TYPE "UDT_ConveyorInterface"
TITLE = UDT_ConveyorInterface
VERSION : 0.1
//User-defined structure of conveyor interface variables.
   STRUCT
      Displacement : Int;   // Displacement per PLC scan [cm] either from position (if available) or speed and time
      SpeedSetpoint : Int;   // Conveyor speed setpoint [mm/s]
      ActualSpeed : Int;   // Conveyors actual speed [mm/s]
      DeltaPosition : Int;   // Read from Conveyor Servo Position [mm] after 1 PLC cycle
      RunFwd { ExternalAccessible := 'False'; ExternalVisible := 'False'; ExternalWritable := 'False'} : Bool;   // Run forward request
      RunRvs { ExternalAccessible := 'False'; ExternalVisible := 'False'; ExternalWritable := 'False'} : Bool;   // Run reverse request
      InternalErrorEncoder { ExternalAccessible := 'False'; ExternalVisible := 'False'; ExternalWritable := 'False'} : Bool;   // Encoder has an error
      InternalErrorVFD { ExternalAccessible := 'False'; ExternalVisible := 'False'; ExternalWritable := 'False'} : Bool;   // VFD has an error
      InternalErrorTracking { ExternalAccessible := 'False'; ExternalVisible := 'False'; ExternalWritable := 'False'} : Bool;   // Tracking has an error
      InternalErrorPEC { ExternalAccessible := 'False'; ExternalVisible := 'False'; ExternalWritable := 'False'} : Bool;   // PEC has an error
      InternalWarningVFD { ExternalAccessible := 'False'; ExternalVisible := 'False'; ExternalWritable := 'False'} : Bool;   // VFD has a warning
      InternalWarningTracking { ExternalAccessible := 'False'; ExternalVisible := 'False'; ExternalWritable := 'False'} : Bool;   // Tracking has a warning
      InternalErrorReset { ExternalAccessible := 'False'; ExternalVisible := 'False'; ExternalWritable := 'False'} : Bool;   // Reset internal errors
      ConfigurationError { ExternalAccessible := 'False'; ExternalVisible := 'False'; ExternalWritable := 'False'} : Bool;   // Configuration error is active
      VFDRunning { ExternalAccessible := 'False'; ExternalVisible := 'False'; ExternalWritable := 'False'} : Bool;   // Motor is running
      VFDatSpeed { ExternalAccessible := 'False'; ExternalVisible := 'False'; ExternalWritable := 'False'} : Bool;   // Motor at speed setpoint
      Disconnected { ExternalAccessible := 'False'; ExternalVisible := 'False'; ExternalWritable := 'False'} : Bool;   // VFD disconnected
      ManualModeActive { ExternalAccessible := 'False'; ExternalVisible := 'False'; ExternalWritable := 'False'} : Bool;   // Covneyor is in manual mode
      ResetStatistics { ExternalAccessible := 'False'; ExternalVisible := 'False'; ExternalWritable := 'False'} : Bool;   // Reset statistics
      HardwareOk { ExternalAccessible := 'False'; ExternalVisible := 'False'; ExternalWritable := 'False'} : Bool;   // Hardware for the Equipment is available and healthy
   END_STRUCT;

END_TYPE

FUNCTION "FC_EquipmentReport" : Void
TITLE = FC_Equipment_Report
{ S7_Optimized_Access := 'TRUE' }
AUTHOR : MHSE
FAMILY : GeneralSystemFunctions
VERSION : 3.0
// ATTRIBUTES
// AUTO_NUMBER = True
// BLOCK_NUMBER = 16
// END_ATTRIBUTES
//Function to generate equipment report.
   VAR_INPUT
      iUDT_Status : "UDT_CommonStatus";   // Status structure
   END_VAR

   VAR_IN_OUT
      iqUDT_Control : "UDT_EquipmentControl";   // Equipment control
   END_VAR


BEGIN
	(*
	----------------------------------------------------------------------------------------

	Version history:
	Date        | Version   | Author        | Remark
	----------------------------------------------------------------------------------------
	24/05/2019  | 0.1       | F.Baten       | first release MHS TIA 15.1
	17/06/2019  | 0.3       | L.Klar        | Manual mode added to "UDT_EquipmentControl"
	17/07/2019  | 0.4       | A.Nowak       | Add all statuses and comments
	24/07/2019  | 2.0       | L.Klar        | 2.0 MHS library release TIA 15.1
	27/08/2019  | 2.1       | K.Pokorski    | Comments adjusted
	16/09/2019  | 2.2       | K.Pokorski    | Equipment error free condition added to "Restart required" status
	06/10/2019  | 2.3       | S. Deukar     | Updated accoring to new UDT equipment report
	12/11/2019  | 3.0       | P.Majka       | 3.0 MHS library release TIA 15.1
	05/02/2024  | 3.1       | L.Klar        | Auto On extention added
	13/03/2024  | 4.0       | S. Nieswiec   | Added to baseline
	*)

	REGION 1 - Equipment report update

	    // Extension of stopped equipment report with the stopped status
	    #iqUDT_Control.Report.Stopped := #iUDT_Status.Stopped
	    OR #iqUDT_Control.Report.Stopped;

	    // Extension of started equipment report with the started status
	    #iqUDT_Control.Report.Running := #iUDT_Status.Running
	    OR #iqUDT_Control.Report.Running;

	    // Extension of energy save equipment report with the energy save status
	    #iqUDT_Control.Report.EnergySave := #iUDT_Status.EnergySave
	    OR #iqUDT_Control.Report.EnergySave;

	    // Extension of warning equipment report with the warning status
	    #iqUDT_Control.Report.Warning := #iUDT_Status.Warning
	    OR #iqUDT_Control.Report.Warning;

	    // Extension of manual mode equipment report with the manual mode status
	    #iqUDT_Control.Report.Manual := #iUDT_Status.Manual
	    OR #iqUDT_Control.Report.Manual;

	    // Extension of error equipment report with the error status
	    #iqUDT_Control.Report.Error := #iUDT_Status.Error
	    OR #iqUDT_Control.Report.Error;

	    // Extension of safety stop equipment report with the safety stop status
	    #iqUDT_Control.Report.SafetyStop := #iUDT_Status.SafetyStop
	    OR #iqUDT_Control.Report.SafetyStop;

	    // Extension of Auto On equipment report with the Auto On status
	    #iqUDT_Control.Report.AutoON := #iUDT_Status.AutoON
	    OR #iqUDT_Control.Report.AutoON;

	    // Extension of restart required equipment report with the restart required and no equipment error statuses
	    #iqUDT_Control.Request.RestartRequired := #iUDT_Status.Stopped
	    AND NOT #iUDT_Status.Error
	    OR #iqUDT_Control.Request.RestartRequired;

	END_REGION
END_FUNCTION

TYPE "UDT_RIOStatistics"
TITLE = UDT_RIOStatistics
VERSION : 0.1
//User-defined structure of FB_RIO function block statistics.
   STRUCT
      PNSlaveNotOnline { S7_SetPoint := 'False'} : "UDT_EventStatistic";   // Statistics of  Profinet slave not online
      PNSlaveError { S7_SetPoint := 'False'} : "UDT_EventStatistic";   // Statistics of a Profinet slave error
   END_STRUCT;

END_TYPE

TYPE "UDT_FlowSplitterCommand"
TITLE = Flow Splitter Command
VERSION : 0.1
   STRUCT
      PercentageSplit : Int;   // Percentage value [%] that diverts are on.
      Mode : Int;   // 1- 100% transport; 2- 50% transport; 3- 100% divert; 4- % divert via HMI; 5- Semi automatic
      ManualMode { ExternalAccessible := 'False'; ExternalVisible := 'False'; ExternalWritable := 'False'} : Bool;   // Manual mode command from HMI
      ManualStartStop { ExternalAccessible := 'False'; ExternalVisible := 'False'; ExternalWritable := 'False'} : Bool;   // Start conveyor running when the bit is true, stop conveyor when the bit is false
      ManualFullSpeed { ExternalAccessible := 'False'; ExternalVisible := 'False'; ExternalWritable := 'False'} : Bool;   // Full speed conveyor in manual mode
      ManualJog { ExternalAccessible := 'False'; ExternalVisible := 'False'; ExternalWritable := 'False'} : Bool;   // Command to jog conveyor in slow speed from HMI
      Zone1DivertActivation { ExternalAccessible := 'False'; ExternalVisible := 'False'; ExternalWritable := 'False'} : Bool;   // Active diverts in zone 1
      Zone2DivertActivation { ExternalAccessible := 'False'; ExternalVisible := 'False'; ExternalWritable := 'False'} : Bool;   // Active diverts in zone 2
   END_STRUCT;

END_TYPE

TYPE "UDT_FlowSplitterStatus"
TITLE = Flow splitter status
VERSION : 0.1
   STRUCT
      Status : Int;   // Status number
      Specific : Struct
         Mode : Int;   // Mode: 1- 100% transport; 2- 50% transport; 3- 100% divert; 4- % divert via HMI; 5- Semi automatic
         Debris { ExternalAccessible := 'False'; ExternalVisible := 'False'; ExternalWritable := 'False'} : Bool;   // Debris detected under the belt
         PEC_EoSJam { ExternalAccessible := 'False'; ExternalVisible := 'False'; ExternalWritable := 'False'} : Bool;   // PEC Jam detected
         PEC_DivertChuteJam { ExternalAccessible := 'False'; ExternalVisible := 'False'; ExternalWritable := 'False'} : Bool;   // PEC divert chute jam detected
         DivertsActivationError { ExternalAccessible := 'False'; ExternalVisible := 'False'; ExternalWritable := 'False'} : Bool;   // Error when zone 1 is not active but zone 2 is active
         AirPressure { ExternalAccessible := 'False'; ExternalVisible := 'False'; ExternalWritable := 'False'} : Bool;   // Air pressure error
         EncoderError { ExternalAccessible := 'False'; ExternalVisible := 'False'; ExternalWritable := 'False'} : Bool;   // Encoder error
         Zone1Divert { ExternalAccessible := 'False'; ExternalVisible := 'False'; ExternalWritable := 'False'} : Bool;   // Zone 1 divert is active
         Zone2Divert { ExternalAccessible := 'False'; ExternalVisible := 'False'; ExternalWritable := 'False'} : Bool;   // Zone 2 divert is active
      END_STRUCT;
   END_STRUCT;

END_TYPE

TYPE "UDT_CaljanReceiveV2"
VERSION : 0.1
   STRUCT
      Healthy { ExternalAccessible := 'False'; ExternalVisible := 'False'; ExternalWritable := 'False'} : Bool;   // True if (un)loader is healthy
      BeltDirection_Loading { ExternalAccessible := 'False'; ExternalVisible := 'False'; ExternalWritable := 'False'} : Bool;   // True if belt is running in loading mode
      BeltDirection_Unloading { ExternalAccessible := 'False'; ExternalVisible := 'False'; ExternalWritable := 'False'} : Bool;   // True if belt is running in unloading mode
      ReadyToReceive { ExternalAccessible := 'False'; ExternalVisible := 'False'; ExternalWritable := 'False'} : Bool;   // True if loader is ready to receive
      ChuteBlockedActivated { ExternalAccessible := 'False'; ExternalVisible := 'False'; ExternalWritable := 'False'} : Bool;   // True when the button chute blocked at the keypad is set
      PECLoader { ExternalAccessible := 'False'; ExternalVisible := 'False'; ExternalWritable := 'False'} : Bool;   // True when no parcels are detected (fail safe) Signal from Caljan Front photo eye
      PECUnloader { ExternalAccessible := 'False'; ExternalVisible := 'False'; ExternalWritable := 'False'} : Bool;   // True when no parcels are detected (fail safe). Signal from Caljan Rear photo eye
      StoreModeActivated { ExternalAccessible := 'False'; ExternalVisible := 'False'; ExternalWritable := 'False'} : Bool;   // True when store mode is selected at the kyepad
      RunModeActivated { ExternalAccessible := 'False'; ExternalVisible := 'False'; ExternalWritable := 'False'} : Bool;   // True when the run mode is selected at the keypad
      LowerOngoing { ExternalAccessible := 'False'; ExternalVisible := 'False'; ExternalWritable := 'False'} : Bool;   // True when the "lower belt" hydraulic valve is active
      RaisingOngoing { ExternalAccessible := 'False'; ExternalVisible := 'False'; ExternalWritable := 'False'} : Bool;   // True when the "raise belt" hydraulic valve is active
      "Spare_I1.3" { ExternalAccessible := 'False'; ExternalVisible := 'False'; ExternalWritable := 'False'} : Bool;   // Spare Bit 3
      "Spare_I1.4" { ExternalAccessible := 'False'; ExternalVisible := 'False'; ExternalWritable := 'False'} : Bool;   // Spare Bit 4
      "Spare_I1.5" { ExternalAccessible := 'False'; ExternalVisible := 'False'; ExternalWritable := 'False'} : Bool;   // Spare Bit 5
      "Spare_I1.6" { ExternalAccessible := 'False'; ExternalVisible := 'False'; ExternalWritable := 'False'} : Bool;   // Spare Bit 6
      "Spare_I1.7" { ExternalAccessible := 'False'; ExternalVisible := 'False'; ExternalWritable := 'False'} : Bool;   // Spare Bit 7
      ActualSpeed : Int;   // Speed in milimeters per second
      Spare_IW4 : Word;   // Spare Word 4
      Spare_IW6 : Word;   // Spare Word 6
   END_STRUCT;

END_TYPE

TYPE "UDT_DimensionsCheckStatus"
VERSION : 0.1
   STRUCT
      Status : Int;   // Status number
      Specific : Struct   // Specific status
         ParcelTooLong { ExternalAccessible := 'False'; ExternalVisible := 'False'; ExternalWritable := 'False'} : Bool;   // Parcel is too long
         ParcelTooHigh { ExternalAccessible := 'False'; ExternalVisible := 'False'; ExternalWritable := 'False'} : Bool;   // Parcel is too high
         ParcelTooWide { ExternalAccessible := 'False'; ExternalVisible := 'False'; ExternalWritable := 'False'} : Bool;   // Parcel is too wide
      END_STRUCT;
   END_STRUCT;

END_TYPE

TYPE "UDT_GateStatus"
VERSION : 0.1
   STRUCT
      Status : Int;   // HMI status structure
      Specific : Struct
         GateClosed { ExternalAccessible := 'False'; ExternalVisible := 'False'; ExternalWritable := 'False'} : Bool;   // When TRUE then gate is closed, when FALSE then gate is open
         GateClosedAndNoOperatorPresent { ExternalAccessible := 'False'; ExternalVisible := 'False'; ExternalWritable := 'False'} : Bool;   // When TRUE then gate is closed, no operator is inside
      END_STRUCT;
   END_STRUCT;

END_TYPE

TYPE "UDT_EmptyWindow"
VERSION : 0.1
   STRUCT
      EmptyWindoSize : Int;   // Minimum size of empty window [mm]
      Last_InductPosition : Int;   // Last inducted position
      No_Of_Empty_Window : Int;   // Number of empty window
      Displacement : Int;   // Displacement [cm/scan]
      EmptyWIndowPosition : Array[0..50] of Int;   // Array of avaiable empty windows
   END_STRUCT;

END_TYPE

TYPE "UDT_CaljanConfigurationV2"
TITLE = UDT_UnloaderConfiguration
VERSION : 0.1
//User-defined structure of unloader parameters.
   STRUCT
      PNDeviceName : String;   // Profinet device Name
      FirstConveyorToStart { ExternalAccessible := 'False'; ExternalVisible := 'False'; ExternalWritable := 'False'} : Bool;   // First conveyor to start cascade mode
      Energy { ExternalAccessible := 'False'; ExternalVisible := 'False'; ExternalWritable := 'False'} : Bool;   // Energy save mode enable
      EnergySaveLenght : DInt;   // Distance conveyor travelled before energy save activate [cm]
      ResetDelay : UDInt := 1000;   // Time required
      CascadeTimeOnDelay : UDInt;   // Cascade time on delay [ms]
      BufferPEC { ExternalAccessible := 'False'; ExternalVisible := 'False'; ExternalWritable := 'False'} : Bool;   // TRUE when buffer PEC from system is available
   END_STRUCT;

END_TYPE

TYPE "UDT_CaljanStatusV2"
TITLE = UDT_UnloaderStatus
VERSION : 0.1
//User-defined structure of FB_Unloader function block status.
   STRUCT
      Status : Int;   // Status number
      Specific : Struct   // Equipment specific warnings and errors
         PEC_EoS : "UDT_PECStatus";   // PEC status structure
         PNSlaveNotOnline { ExternalAccessible := 'False'; ExternalVisible := 'False'; ExternalWritable := 'False'} : Bool;   // Profinet slave is not online
         PNSlaveError { ExternalAccessible := 'False'; ExternalVisible := 'False'; ExternalWritable := 'False'} : Bool;   // Profinet slave is in error
         PNSlaveWarning { ExternalAccessible := 'False'; ExternalVisible := 'False'; ExternalWritable := 'False'} : Bool;   // Profinet slave has  a warning
         Disabled { ExternalAccessible := 'False'; ExternalVisible := 'False'; ExternalWritable := 'False'} : Bool;   // Unloader is disabled by HMI
         VFDError { ExternalAccessible := 'False'; ExternalVisible := 'False'; ExternalWritable := 'False'} : Bool;   // Unloader has an VFD error
         NotHealthy { ExternalAccessible := 'False'; ExternalVisible := 'False'; ExternalWritable := 'False'} : Bool;   // Unloader is not healthy
         StoreMode { ExternalAccessible := 'False'; ExternalVisible := 'False'; ExternalWritable := 'False'} : Bool;   // Store mode activated
         RunMode { ExternalAccessible := 'False'; ExternalVisible := 'False'; ExternalWritable := 'False'} : Bool;   // Run mode activated
         LowerOngoing { ExternalAccessible := 'False'; ExternalVisible := 'False'; ExternalWritable := 'False'} : Bool;   // "lower belt" hydraulic valve is active
         RaisingOngoing { ExternalAccessible := 'False'; ExternalVisible := 'False'; ExternalWritable := 'False'} : Bool;   // "raise belt" hydraulic valve is active
         ChuteBlocked { ExternalAccessible := 'False'; ExternalVisible := 'False'; ExternalWritable := 'False'} : Bool;   // Chute blocked activated
      END_STRUCT;
   END_STRUCT;

END_TYPE

TYPE "UDT_CaljanSendV2"
VERSION : 0.1
   STRUCT
      Enable { ExternalAccessible := 'False'; ExternalVisible := 'False'; ExternalWritable := 'False'} : Bool;   // Needs to be True for the “Run” mode to be active
      AllowLoading { ExternalAccessible := 'False'; ExternalVisible := 'False'; ExternalWritable := 'False'} : Bool;   // True if belt start in loading mode is allowed
      AllowUnloading { ExternalAccessible := 'False'; ExternalVisible := 'False'; ExternalWritable := 'False'} : Bool;   // True if belt start in unloading mode is allowed
      Reset { ExternalAccessible := 'False'; ExternalVisible := 'False'; ExternalWritable := 'False'} : Bool;   // Reset error and safety command
      BufferPEC { ExternalAccessible := 'False'; ExternalVisible := 'False'; ExternalWritable := 'False'} : Bool;   // Photoeye signal. Used for store mode. True when product is detected.
      "Spare_Q0.5" { ExternalAccessible := 'False'; ExternalVisible := 'False'; ExternalWritable := 'False'} : Bool;   // Spare Bit 5
      JogReverseCommand { ExternalAccessible := 'False'; ExternalVisible := 'False'; ExternalWritable := 'False'} : Bool;   // While TRUE the extendible conveyor should run in reverse (external hold-to-run reverse signal) Reverse = Loading direction
      "Spare_Q0.7" { ExternalAccessible := 'False'; ExternalVisible := 'False'; ExternalWritable := 'False'} : Bool;   // Spare Bit 7
      Spare_QB1 : Byte;   // Spare Byte 1
      Spare_QW2 : Word;   // Spare Word 2
      Spare_QW4 : Word;   // Spare Word 4
      Spare_QW6 : Word;   // Spare Word 6
   END_STRUCT;

END_TYPE

TYPE "UDT_CaljanStatisticsV2"
TITLE = UDT_UnloaderStatistics
VERSION : 0.1
//User-defined structure of FB_Unloader function block statistics.
   STRUCT
      EnergySave : "UDT_EventStatistic";   // Number of times that save energy mode occurs
      ExtendableUpTime : "UDT_EventStatistic";   // Conveyor up time
      ExtendableDownTime : "UDT_EventStatistic";   // Conveyor down time
      VFDError : "UDT_EventStatistic";   // VFD Error
      NotHealthy : "UDT_EventStatistic";   // Extendable not healthy
      PEC_EOS : "UDT_PECStatistics";   // PEC error
      PNNodeNotOnline : "UDT_EventStatistic";   // PN node not online
      PNNodeError : "UDT_EventStatistic";   // PN node has error
   END_STRUCT;

END_TYPE

TYPE "UDT_HS10080XCTConfiguration"
VERSION : 0.1
   STRUCT
      InfeedConveyor : "UDT_ConveyorCommonConfiguration";
      MainConveyor : "UDT_ConveyorCommonConfiguration";
      OutfeedConveyor : "UDT_ConveyorCommonConfiguration";
      PEC_InfeedTimeOnDelay : UDInt;   // Photo eye time on delay [ms]
      PEC_InfeedTimeOffDelay : UDInt;   // Photo eye time off delay [ms]
      PEC_InfeedDistance : Int;   // Distance between photo eye and the end of conveyor [mm]
      PEC_InfeedDistanceOffset : Int;   // Distance offset between photo eye and the end of conveyor [mm]
      PEC_OutfeedTimeOnDelay : UDInt;   // Photo eye time on delay [ms]
      PEC_OutfeedTimeOffDelay : UDInt;   // Photo eye time off delay [ms]
      PEC_OutfeedDistance : Int;   // Distance between photo eye and the end of conveyor [mm]
      PEC_OutfeedDistanceOffset : Int;   // Distance offset between photo eye and the end of conveyor [mm]
      OutfeedPECJamDisplacementLimit : Int;   // Limit displacement with PEC blocked to detect jam [cm]
      InfeedPECJamDisplacementLimit : Int;   // Limit displacement with PEC blocked to detect jam [cm]
      Gap : Int;   // Gapping tail to head value [cm]
      CallibrationTimeout : UDInt;   // Max time when callibration is requested before "ix_AllowCallibration" is overruled
      MainConvFeedbackDelayTime : UInt;   // Time limit to check XRAY main conveyor speed OK feedback (ms)
      EnergySaveLenght : Int;   // Distance conveyor travelled before energy save activate [cm]
      CascadeTimeOnDelay : UDInt;   // Cascade time on delay [ms]
      Energy { ExternalAccessible := 'False'; ExternalVisible := 'False'; ExternalWritable := 'False'} : Bool;   // Energy save mode enable
      FirstConveyorToStart { ExternalAccessible := 'False'; ExternalVisible := 'False'; ExternalWritable := 'False'} : Bool;   // First conveyor to start cascade mode
      ResetWithPECBlocked { ExternalAccessible := 'False'; ExternalVisible := 'False'; ExternalWritable := 'False'} : Bool;   // When 'True' - Allow reset system after jam with the PEC blocked
   END_STRUCT;

END_TYPE

TYPE "UDT_HS10080XCTHMICommand"
VERSION : 0.1
   STRUCT
      NoScanMode { ExternalAccessible := 'False'; ExternalVisible := 'False'; ExternalWritable := 'False'} : Bool;   // NO scan mode command from HMI
   END_STRUCT;

END_TYPE

TYPE "UDT_FlowSplitterConfiguration"
TITLE = Flow Splitter Configuration
VERSION : 0.1
   STRUCT
      PEC_EoSTimeOnDelay : UDInt;   // Photo eye time on delay [ms]
      PEC_EoSTimeOffDelay : UDInt;   // Photo eye time off delay [ms]
      PEC_FilterChuteTimeOnDelay : UDInt;   // Divert chute photo eye time on delay [ms]
      PEC_FilterChuteTimeOffDelay : UDInt;   // Divert chute photo eye time off delay [ms]
      PEC_FilterUpstreamTimeOnDelay : UDInt;   // Upstream photo eye time on delay [ms]
      PEC_FilterUpstreamTimeOffDelay : UDInt;   // Upstream photo eye time off delay [ms]
      AirPressure_FilterTimeOffDelay : UDInt;   // Air pressure time off delay [ms]
      DivertsTimeActivation : UDInt;   // Time to enable diverts pop-up [ms]
      CascadeTimeOnDelay : UDInt;   // Cascade time on delay [ms]
      DebrisTimeFilter : UDInt;   // Time to filter debris sensor signal [ms]
      SpeedSetpointNominal : Int;   // Nominal speed setpoint [mm/s]
      SpeedSetpointLow : Int;   // Low speed setpoint [mm/s]
      DivertSwitchDelay : Int;   // Divert switch delay [s]
      JamDisplacementLimit : Int;   // Limit displacement with PEC blocked to detect jam [cm]
      DivertChuteJamDisplacLimit : Int;   // Limit displacement with PEC divert chute blocked to detect jam [cm]
      TimeBasedSplit : Int;   // Time based split [s]
      Length : Int;   // Conveyor length [mm]
      LengthCorrection : Int;   // Length correction [mm]
      DefaultMode : Int;   // Mode: 1- 100% transport; 2- 50% transport; 3- 100% divert; 4- % divert; 5 - Semi automatic
      PEC_Present { ExternalAccessible := 'False'; ExternalVisible := 'False'; ExternalWritable := 'False'} : Bool;   // Thue when a photo eye is present in the flow splitter
      PEC_ChutePesent { ExternalAccessible := 'False'; ExternalVisible := 'False'; ExternalWritable := 'False'} : Bool;   // Thue when a photo eye is present in the chute
      FirstConveyorToStart { ExternalAccessible := 'False'; ExternalVisible := 'False'; ExternalWritable := 'False'} : Bool;   // First conveyor to start cascade mode
      OnFlyChangeOfMode { ExternalAccessible := 'False'; ExternalVisible := 'False'; ExternalWritable := 'False'} : Bool;   // On fly change of mode
      DivertsTimeSave { ExternalAccessible := 'False'; ExternalVisible := 'False'; ExternalWritable := 'False'} : Bool;   // Disable diverts if there is no parcels
      Energy { ExternalAccessible := 'False'; ExternalVisible := 'False'; ExternalWritable := 'False'} : Bool;   // Energy save mode enable
      EnergySaveLength { ExternalAccessible := 'False'; ExternalVisible := 'False'; ExternalWritable := 'False'} : Int;   // Distance conveyor travelled before energy save activate [cm]
   END_STRUCT;

END_TYPE

TYPE "UDT_CapacityConfiguration"
VERSION : 0.1
   STRUCT
      AveragePackageLengthConfiguration : Int;   // Average package length [mm]
      Interval : UDInt;   // Interval time [s]
      Treshold : Int;   // Minimum value for the capacity to be saved
   END_STRUCT;

END_TYPE

TYPE "UDT_Chute2PECConfiguration"
VERSION : 0.1
//User-defined structure of FB_Chute2PEC function block configuration.
   STRUCT
      FullDetectionTime : UDInt;   // Time after which chute full is detected
      FullReleaseTime : UDInt;   // Time after which chute full is released
      HalfFullDetectionTime : UDInt;   // Time after which chute half full is detected
      HalfFullReleaseTime : UDInt;   // Time after which chute half full is released
   END_STRUCT;

END_TYPE

TYPE "UDT_Chute1PECStatus"
VERSION : 0.1
//User-defined structure of FB_Chute1PEC function block status.
   STRUCT
      Status : Int;   // Status number
      Specific : Struct   // CH02 specific status structure
         ChuteFull { ExternalAccessible := 'False'; ExternalVisible := 'False'; ExternalWritable := 'False'} : Bool;   // Chute is full status
         ChuteDisabled { ExternalAccessible := 'False'; ExternalVisible := 'False'; ExternalWritable := 'False'} : Bool;   // Chute is disabled status
      END_STRUCT;
   END_STRUCT;

END_TYPE

TYPE "UDT_DimensionsCheckStatistics"
VERSION : 0.1
   STRUCT
      TooLongParcels : "UDT_EventStatistic";
      TooHighParcels : "UDT_EventStatistic";
      TooWideParcels : "UDT_EventStatistic";
   END_STRUCT;

END_TYPE

TYPE "UDT_HS10080XCTStatus"
TITLE = UDT_HS10080XCTStatus
VERSION : 0.1
//User-defined structure of FB_Xray_HS10080XCT function block status.
   STRUCT
      Status : Int;   // Status number
      XraySpecific : Struct   // Equipment specific warnings and errors
         XrayPowerNotOn { ExternalAccessible := 'False'; ExternalVisible := 'False'; ExternalWritable := 'False'} : Bool;   // X-ray not turned on
         MachineNotOk { ExternalAccessible := 'False'; ExternalVisible := 'False'; ExternalWritable := 'False'} : Bool;   // X-ray not initialised or not working properly
         XRayNotReady { ExternalAccessible := 'False'; ExternalVisible := 'False'; ExternalWritable := 'False'} : Bool;   // X-ray not ready to receive a bag
         TransitActive { ExternalAccessible := 'False'; ExternalVisible := 'False'; ExternalWritable := 'False'} : Bool;   // Transit mode is active
         NoScanActive { ExternalAccessible := 'False'; ExternalVisible := 'False'; ExternalWritable := 'False'} : Bool;   // X-ray is in the no-scan mode
         IQTestActive { ExternalAccessible := 'False'; ExternalVisible := 'False'; ExternalWritable := 'False'} : Bool;   // IQ test is active on XRAY
         DoorInterlockNotOk { ExternalAccessible := 'False'; ExternalVisible := 'False'; ExternalWritable := 'False'} : Bool;   // One of the doors of the in- or outfeed tunnel is opend
         RepairSwitch { ExternalAccessible := 'False'; ExternalVisible := 'False'; ExternalWritable := 'False'} : Bool;   // X-ray mains are powered off
         ServiceMode { ExternalAccessible := 'False'; ExternalVisible := 'False'; ExternalWritable := 'False'} : Bool;   // X-ray is in service mode.
         TempOutOfRange { ExternalAccessible := 'False'; ExternalVisible := 'False'; ExternalWritable := 'False'} : Bool;   // XCT operating temperature is out of range
         GantrySpeedNotOk { ExternalAccessible := 'False'; ExternalVisible := 'False'; ExternalWritable := 'False'} : Bool;   // Gantry speed is not ok
      END_STRUCT;
      InfeedConvSpecific : Struct   // Equipment specific warnings and errors
         Status : Int;   // Satus number
         Conv_ERR { ExternalAccessible := 'False'; ExternalVisible := 'False'; ExternalWritable := 'False'} : Bool;   // Conveyor is in error
         Encoder_ERR { ExternalAccessible := 'False'; ExternalVisible := 'False'; ExternalWritable := 'False'} : Bool;   // Encoder error
         PEC_EoSJam { ExternalAccessible := 'False'; ExternalVisible := 'False'; ExternalWritable := 'False'} : Bool;   // PE Jammed end of system pec
      END_STRUCT;
      MainConvSpecific : Struct   // Equipment specific warnings and errors
         Status : Int;   // Satus number
         Conv_ERR { ExternalAccessible := 'False'; ExternalVisible := 'False'; ExternalWritable := 'False'} : Bool;   // Conveyor is in error
         Encoder_ERR { ExternalAccessible := 'False'; ExternalVisible := 'False'; ExternalWritable := 'False'} : Bool;   // Encoder error
      END_STRUCT;
      OutfeedConvSpecific : Struct   // Equipment specific warnings and errors
         Status : Int;   // Satus number
         Conv_ERR { ExternalAccessible := 'False'; ExternalVisible := 'False'; ExternalWritable := 'False'} : Bool;   // Conveyor is in error
         Encoder_ERR { ExternalAccessible := 'False'; ExternalVisible := 'False'; ExternalWritable := 'False'} : Bool;   // Encoder error
         PEC_EoSJam { ExternalAccessible := 'False'; ExternalVisible := 'False'; ExternalWritable := 'False'} : Bool;   // PE Jammed end of system pec
      END_STRUCT;
   END_STRUCT;

END_TYPE

TYPE "UDT_DimensionsCheckConfiguration"
VERSION : 0.1
   STRUCT
      DistanceBetweenLenghtPECs : UInt;   // Distance between two Lenght PECs [cm]
      ParcelLengthAllowedDeviation : UInt;   // Maximum torelance in measured parcel length [cm]
      PECLength1OnTime : UDInt;   // Lenght 1 photo eye time on delay [ms]
      PECLength1OffTime : UDInt;   // Lenght 1 photo eye time off delay [ms]
      PECLength2OnTime : UDInt;   // Lenght 2 photo eye time on delay [ms]
      PECLength2OffTime : UDInt;   // Lenght 2 photo eye time off delay [ms]
      PECLength2CheckLimit : UDInt;   // maximum length for length check PEC 2
      PECWidthOnTime : UDInt;   // Width 1 photo eye time on delay [ms]
      PECWidthOffTime : UDInt;   // Width 1 photo eye time off delay [ms]
      PECWidthCheckLimit : UDInt;   // maximum width for width check PEC
      PECHeightTimeOn : UDInt;   // Height photo eye time on delay [ms]
      PECHeightTimeOff : UDInt;   // Height photo eye time off delay [ms]
      AllowedPackageWidth : UInt;   // Maximum package width measured by mode 2
   END_STRUCT;

END_TYPE

TYPE "UDT_DimensionsCheckStatisticsV2"
VERSION : 0.1
   STRUCT
      TooLongParcels : "UDT_EventStatistic";
      TooShortParcels : "UDT_EventStatistic";
      TooHighParcels : "UDT_EventStatistic";
      TooLowParcels : "UDT_EventStatistic";
      TooWideParcels : "UDT_EventStatistic";
      TooNarrowParcels : "UDT_EventStatistic";
      IncorrectShape : "UDT_EventStatistic";
      GeneralError : "UDT_EventStatistic";
   END_STRUCT;

END_TYPE

TYPE "UDT_DimensionsCheckHMIDataV2"
VERSION : 0.1
   STRUCT
      ActualSensor1 : UInt;   // Actual sensor value
      OffsetSensor1 : UInt;   // Sensor offset value
      PositionSensor1 : UInt;   // The value of the sensor after subtracting the offset
      ActualSensor2 : UInt;   // Actual sensor value
      OffsetSensor2 : UInt;   // Sensor offset value
      PositionSensor2 : UInt;   // The value of the sensor after subtracting the offset
      BeltWidth : UInt;   // Belt width
      ProductWidth : UInt;   // Product width
   END_STRUCT;

END_TYPE

TYPE "UDT_DimensionsCheckStatusV2"
VERSION : 0.1
   STRUCT
      Status : Int;   // Status number
      Specific : Struct   // Specific status
         ParcelTooLongError { ExternalAccessible := 'False'; ExternalVisible := 'False'; ExternalWritable := 'False'} : Bool;   // Error - parcel is too long
         ParcelTooShortError { ExternalAccessible := 'False'; ExternalVisible := 'False'; ExternalWritable := 'False'} : Bool;   // Error - parcel is too short
         ParcelTooHighError { ExternalAccessible := 'False'; ExternalVisible := 'False'; ExternalWritable := 'False'} : Bool;   // Error - parcel is too high
         ParcelTooLowError { ExternalAccessible := 'False'; ExternalVisible := 'False'; ExternalWritable := 'False'} : Bool;   // Error - parcel is too low
         ParcelTooWideError { ExternalAccessible := 'False'; ExternalVisible := 'False'; ExternalWritable := 'False'} : Bool;   // Error - parcel is too wide
         ParcelTooNarrowError { ExternalAccessible := 'False'; ExternalVisible := 'False'; ExternalWritable := 'False'} : Bool;   // Error - parcel is too narrow
         IncorrectParcelOrientationError { ExternalAccessible := 'False'; ExternalVisible := 'False'; ExternalWritable := 'False'} : Bool;   // Error - Incorrect parcel orientation
         GeneralError { ExternalAccessible := 'False'; ExternalVisible := 'False'; ExternalWritable := 'False'} : Bool;   // General error
         DisabledGeneralFunctionality { ExternalAccessible := 'False'; ExternalVisible := 'False'; ExternalWritable := 'False'} : Bool;   // Disabled general DMC functionality
         DisabledTooLongParcel { ExternalAccessible := 'False'; ExternalVisible := 'False'; ExternalWritable := 'False'} : Bool;   // Disabled "TooLongParcel" detection
         DisabledTooShortParcelError { ExternalAccessible := 'False'; ExternalVisible := 'False'; ExternalWritable := 'False'} : Bool;   // Disabled "TooShortParcel" detection
         DisabledTooHighParcelError { ExternalAccessible := 'False'; ExternalVisible := 'False'; ExternalWritable := 'False'} : Bool;   // Disabled "TooHighParcel" detection
         DisabledTooLowParcelError { ExternalAccessible := 'False'; ExternalVisible := 'False'; ExternalWritable := 'False'} : Bool;   // Disabled "TooLowParcel" detection
         DisabledTooWideParcelError { ExternalAccessible := 'False'; ExternalVisible := 'False'; ExternalWritable := 'False'} : Bool;   // Disabled "TooWideParcel" detection
         DisabledTooNarrowParcelError { ExternalAccessible := 'False'; ExternalVisible := 'False'; ExternalWritable := 'False'} : Bool;   // Disabled "TooNarrowParcel" detection
         DisabledParcelOrientationError { ExternalAccessible := 'False'; ExternalVisible := 'False'; ExternalWritable := 'False'} : Bool;   // Disabled "ParcelOrientation" detection
      END_STRUCT;
   END_STRUCT;

END_TYPE

TYPE "UDT_DimensionsCheckCommandV2"
TITLE = Flow Splitter Command
VERSION : 0.1
   STRUCT
      DisableGeneral { ExternalAccessible := 'False'; ExternalVisible := 'False'; ExternalWritable := 'False'} : Bool;   // Disable genneral functionality DMC
      DisableTooLongParcelError { ExternalAccessible := 'False'; ExternalVisible := 'False'; ExternalWritable := 'False'} : Bool;   // Disable "TooLongParcel" error
      DisableTooShortParcelError { ExternalAccessible := 'False'; ExternalVisible := 'False'; ExternalWritable := 'False'} : Bool;   // Disable "TooShortParcel" error
      DisableTooHighParcelError { ExternalAccessible := 'False'; ExternalVisible := 'False'; ExternalWritable := 'False'} : Bool;   // Disable "TooHighParcel" error
      DisableTooLowParcelError { ExternalAccessible := 'False'; ExternalVisible := 'False'; ExternalWritable := 'False'} : Bool;   // Disable "TooLowParcel" error
      DisableTooWideParcelError { ExternalAccessible := 'False'; ExternalVisible := 'False'; ExternalWritable := 'False'} : Bool;   // Disable "TooWideParcel" error
      DisableTooNarrowParcelError { ExternalAccessible := 'False'; ExternalVisible := 'False'; ExternalWritable := 'False'} : Bool;   // Disable "TooNarrowParcel" error
      DisableParcelOrientationError { ExternalAccessible := 'False'; ExternalVisible := 'False'; ExternalWritable := 'False'} : Bool;   // Disable "ParcelOrientation" error
      ButtonOffsetDistanceSensor1 { ExternalAccessible := 'False'; ExternalVisible := 'False'; ExternalWritable := 'False'} : Bool;   // Button to set offset value
      ButtonOffsetDistanceSensor2 { ExternalAccessible := 'False'; ExternalVisible := 'False'; ExternalWritable := 'False'} : Bool;   // Button to set offset value
   END_STRUCT;

END_TYPE

TYPE "UDT_Chute1PECStatistics"
VERSION : 0.1
//User-defined structure of FB_Chute1PEC function block statistics.
   STRUCT
      ChuteFull { S7_SetPoint := 'False'} : "UDT_EventStatistic";   // Chute full statistics
      ChuteDisabled { S7_SetPoint := 'False'} : "UDT_EventStatistic";   // Chute disabled statistics
   END_STRUCT;

END_TYPE

TYPE "UDT_DimensionsCheckConfigurationV2"
VERSION : 0.1
   STRUCT
      PEC_Time_Delay : Struct   // Times for sensors ON/OFF delay
         On_MinHeight : UDInt := 30;   // Minimum Height photo eye time on delay [ms]
         Off_MinHeight : UDInt := 30;   // MinimumHeight photo eye time off delay [ms]
      END_STRUCT;
      Position : Struct   // This values is calculeted from the PEC1 to the next one
         MinHeightPEC_Array : Int;   // Distance between Lenght PEC Laser and Min Height PEC Array [mm]
         Width_Distance_Sensor_1 : Int;   // Distance between Lenght PEC Laser and Distance sensor 1 [mm]
         Width_Distance_Sensor_2 : Int;   // Distance between Lenght PEC Laser and Distance sensor 2 [mm]
         BeltWidth : Int;   // Distance between side guards [mm]
      END_STRUCT;
      Limit : Struct   // Limits for parcel size
         MinWidth : Int := 100;   // Minimum width [mm]
         MaxWidth : Int := 900;   // Maximum width [mm]
         MinLength : Int := 100;   // Minimum length [mm]
         MaxLength : Int := 1200;   // Maximum length [mm]
         TooHighDistance : Int := 200;   // Distance [mm]
         TooLongDistance : Int := 1400;   // Distance [mm]
      END_STRUCT;
      Tolerance : Struct   // Tolerance for parcel size
         TooWide : Int;   // [%] - Percentage of deviations
         TooNarrow : Int;   // [%] - Percentage of deviations
         TooHigh : Int;   // [%] - Percentage of deviations
         TooLow : Int;   // [%] - Percentage of deviations
         Orientation : Int;   // [%] - Percentage of deviations
      END_STRUCT;
      Functionality : Struct   // Set TRUE if functionality should be enabled
         TooLongParcelError { ExternalAccessible := 'False'; ExternalVisible := 'False'; ExternalWritable := 'False'} : Bool;   // If true "TooLongParcel"detection active
         TooShortParcelError { ExternalAccessible := 'False'; ExternalVisible := 'False'; ExternalWritable := 'False'} : Bool;   // If true "TooShortParcel"detection active
         TooHighParcelError { ExternalAccessible := 'False'; ExternalVisible := 'False'; ExternalWritable := 'False'} : Bool;   // If true "TooHighParcel"detection active
         TooLowParcelError { ExternalAccessible := 'False'; ExternalVisible := 'False'; ExternalWritable := 'False'} : Bool;   // If true "TooLowParcel"detection active
         TooWideParcelError { ExternalAccessible := 'False'; ExternalVisible := 'False'; ExternalWritable := 'False'} : Bool;   // If true "TooWideParcel"detection active
         TooNarrowParcelError { ExternalAccessible := 'False'; ExternalVisible := 'False'; ExternalWritable := 'False'} : Bool;   // If true "TooNarrowParcel"detection active
         ParcelOrientationError { ExternalAccessible := 'False'; ExternalVisible := 'False'; ExternalWritable := 'False'} : Bool;   // If true "ParcelOrientation"detection active
      END_STRUCT;
   END_STRUCT;

END_TYPE

TYPE "UDT_ControlPowerGroupWORStatus"
VERSION : 0.1
   STRUCT
      Status : Int;   // Status number
      Specific : Struct
         PowerSuppliesError { ExternalAccessible := 'False'; ExternalVisible := 'False'; ExternalWritable := 'False'} : Bool;   // Power supplly error
      END_STRUCT;
   END_STRUCT;

END_TYPE

TYPE "UDT_FlowSplitterStatistics"
TITLE = Flow splitter statistics
VERSION : 0.1
   STRUCT
      FlowSplitterUpTime : "UDT_EventStatistic";   // Flow splitter up time
      FlowSplitterDownTime : "UDT_EventStatistic";   // Flow splitter down time
      PECChuteDivertJam : "UDT_EventStatistic";   // PEC chute divert jam
      PEC_EoSJam : "UDT_EventStatistic";   // PEC end of section jam
      AirPressure : "UDT_EventStatistic";   // Air pressure fault
      DebrisSensor : "UDT_EventStatistic";   // Debris detected under the belt
      EncoderError : "UDT_EventStatistic";   // Encoder error
      Mode100Straight : "UDT_EventStatistic";   // 100% send to straight downstream conveyor
      "Mode50/50" : "UDT_EventStatistic";   // 50% send to straight downstream conveyor, 50% send to divert downstream conveyor
      Mode100Divert : "UDT_EventStatistic";   // 100% send to divert downstream conveyor
      ModeTimeBasedSplit : "UDT_EventStatistic";   // Time base split mode
      ModeSemiAutomatic : "UDT_EventStatistic";   // Semi automatic mode
      EnergySave : "UDT_EventStatistic";   // Number of times that save energy mode occurs
   END_STRUCT;

END_TYPE

TYPE "UDT_ControlPowerGroupWORStatistics"
VERSION : 0.1
   STRUCT
      PowerSupplyError : "UDT_EventStatistic";   // Error Power Supply Group Statistics
   END_STRUCT;

END_TYPE

TYPE "UDT_ConnectStatus"
VERSION : 0.1
   STRUCT
      Status : Int;   // Status number
      Specific : Struct   // Specific status structure
         Connected { ExternalAccessible := 'False'; ExternalVisible := 'False'; ExternalWritable := 'False'} : Bool;   // Connected
         CommunicationFault { ExternalAccessible := 'False'; ExternalVisible := 'False'; ExternalWritable := 'False'} : Bool;   // Communication fault
      END_STRUCT;
   END_STRUCT;

END_TYPE

TYPE "UDT_Chute2PECStatus"
VERSION : 0.1
//User-defined structure of FB_CH03 function block status.
   STRUCT
      Status : Int;   // Status number
      Specific : Struct   // CH02 specific status structure
         ChuteFull { ExternalAccessible := 'False'; ExternalVisible := 'False'; ExternalWritable := 'False'} : Bool;   // Chute is full status
         ChuteHalfFull { ExternalAccessible := 'False'; ExternalVisible := 'False'; ExternalWritable := 'False'} : Bool;   // Chute is half full status
         ChuteDisabled { ExternalAccessible := 'False'; ExternalVisible := 'False'; ExternalWritable := 'False'} : Bool;   // Chute is disabled status
      END_STRUCT;
   END_STRUCT;

END_TYPE

TYPE "UDT_Chute2PECStatistics"
VERSION : 0.1
//User-defined structure of FB_CH03 function block statistics.
   STRUCT
      ChuteFull { S7_SetPoint := 'False'} : "UDT_EventStatistic";   // Chute full statistics
      ChuteHalfFull : "UDT_EventStatistic";   // Chute half full statistics
      ChuteDisabled { S7_SetPoint := 'False'} : "UDT_EventStatistic";   // Chute disabled statistics
   END_STRUCT;

END_TYPE

TYPE "UDT_Chute1PECConfiguration"
VERSION : 0.1
//User-defined structure of FB_Chute1PEC function block configuration.
   STRUCT
      FullDetectionTime : UDInt;   // Time after which chute full is detected
      FullReleaseTime : UDInt;   // Time after which chute full is released
   END_STRUCT;

END_TYPE

TYPE "UDT_EuchnerLockStatus"
VERSION : 0.1
   STRUCT
      LockFault { ExternalAccessible := 'False'; ExternalVisible := 'False'; ExternalWritable := 'False'} : Bool;   // Internal lock fault
      DoorClosed { ExternalAccessible := 'False'; ExternalVisible := 'False'; ExternalWritable := 'False'} : Bool;   // The door is closed
      DoorOpened { ExternalAccessible := 'False'; ExternalVisible := 'False'; ExternalWritable := 'False'} : Bool;   // The door is opened
      BoltTongueClosed { ExternalAccessible := 'False'; ExternalVisible := 'False'; ExternalWritable := 'False'} : Bool;   // The lock bolt tongue is closed
      Safelylocked { ExternalAccessible := 'False'; ExternalVisible := 'False'; ExternalWritable := 'False'} : Bool;   // The lock is safely locked
      SafetyLockAckReq { ExternalAccessible := 'False'; ExternalVisible := 'False'; ExternalWritable := 'False'} : Bool;   // The safety lock signal needs to be confirmed
   END_STRUCT;

END_TYPE

TYPE "UDT_HS10080XCTStatistics"
TITLE = UDT_HS10080XCTStatistics
VERSION : 0.1
//User-defined structure of FB_Xray_HS10080XCT function block statistics.
   STRUCT
      XRayMode : "UDT_EventStatistic";   // Running in X-Ray mode
      ServiceMode : "UDT_EventStatistic";   // Running in service mode
      TransitMode : "UDT_EventStatistic";   // Running in transit mode
      EStopActive : "UDT_EventStatistic";   // E-Stop is active
      RepairSwitch : "UDT_EventStatistic";   // Mains power on
      TempOutOfRange : "UDT_EventStatistic";   // XCT doesn’t work because XCT operating temperature isn’t given.
      Stopped : "UDT_EventStatistic";   // Machine is stopped
      Calibrating : "UDT_EventStatistic";   // Calibration is active
      CallibrationForced : "UDT_EventStatistic";   // Callibration is forced on (timed out waiting)
      Interlock : "UDT_EventStatistic";   // One of the doors of the in or outfeed tunnel is opend
      InfeedConveyorError : "UDT_EventStatistic";   // The Infeed conveyor was in error
      OutfeedConveyorError : "UDT_EventStatistic";   // The Outfeed conveyor was in error
      EncoderError : "UDT_EventStatistic";   // One of the encoders has faulted
   END_STRUCT;

END_TYPE

TYPE "UDT_VfdPositioningStatus"
TITLE = UDT_VfdPositioningStatus
VERSION : 0.1
//User-defined structure of VFD SEW positioning status.
   STRUCT
      ErrorCode : Int;   // Error code
      SubErrorCode : Int;   // Sub error code
      PNSlaveNotOnline : Bool := FALSE;   // Profinet slave is not on line
      PNSlaveError : Bool := FALSE;   // Profinet slave has an error
      InternalError : Bool := FALSE;   // A VFD internal error is active, see error code
      InternalWarning : Bool := FALSE;   // A VFD internal warning is active, see error code
      CommunicationErrorMovikit : Bool := FALSE;   // Communication error with MoviKit
      PositioningTimeOutError : Bool := FALSE;   // Exceeded time to reach position
      PNSlaveWarning { ExternalAccessible := 'False'; ExternalVisible := 'False'; ExternalWritable := 'False'} : Bool;   // Profinet slave has a warning
   END_STRUCT;

END_TYPE

TYPE "UDT_XBSInductInterfaceSend"
VERSION : 0.1
   STRUCT
      WatchDog : Byte;   // Watch dog counter
      IncomingParcel { ExternalAccessible := 'False'; ExternalVisible := 'False'; ExternalWritable := 'False'} : Bool;   // Parcel found in 2-meter distance from the induct line
      Discharge { ExternalAccessible := 'False'; ExternalVisible := 'False'; ExternalWritable := 'False'} : Bool;   // Transfer in Progress
      ParcelOnBoard : DInt;   // Number of parcels in 2-meter distance from the induct line
      ParcelID : DInt;   // ParcelID of the parcel in transfer
      ObjectID : DInt;   // ObjectID Of the parcel in the transfer
      LastConveyorSpeed : Real;   // Actual speed of the last conveyor (mm/sec)
   END_STRUCT;

END_TYPE

TYPE "UDT_Induct"
VERSION : 0.1
   STRUCT
      DistanceLastReserved { S7_SetPoint := 'True'} : Int;   // The distance after which the next window will be reserved
      DisableWindowReservation { ExternalAccessible := 'False'; ExternalVisible := 'False'; ExternalWritable := 'False'} : Bool;   // Signal to disable window reservation
      AutoRecovery { ExternalAccessible := 'False'; ExternalVisible := 'False'; ExternalWritable := 'False'} : Bool;   // Signal for induct to auto recover
      Position : Array[1..20] of "UDT_InductParcelData";   // Position
   END_STRUCT;

END_TYPE

TYPE "UDT_InductConfiguration"
VERSION : 0.1
   STRUCT
      Induct_Number { ExternalAccessible := 'False'; ExternalVisible := 'False'; ExternalWritable := 'False'} : Int := 1;   // Induct number where the most upstream induct is 1
      Induct_Position { ExternalAccessible := 'False'; ExternalVisible := 'False'; ExternalWritable := 'False'} : Int := 100;   // Virtual position of the induct [mm] on the merge tracking DB
      GapMode { ExternalAccessible := 'False'; ExternalVisible := 'False'; ExternalWritable := 'False'} : Int := 2;   // 1=HeadToHead, 2=Length+fixedgap size 3=Length+flex gapsize
      GapHeadToHead { ExternalAccessible := 'False'; ExternalVisible := 'False'; ExternalWritable := 'False'} : Int := 150;   // Gapping head to head value [cm]
      GapTailToHead { ExternalAccessible := 'False'; ExternalVisible := 'False'; ExternalWritable := 'False'} : Int := 10;   // Gapping tail to head value [cm]
      MaxParcelSize { ExternalAccessible := 'False'; ExternalVisible := 'False'; ExternalWritable := 'False'} : Int := 30;   // Maximum size parcel [mm] to set when no size is found
      MinParcelSize { ExternalAccessible := 'False'; ExternalVisible := 'False'; ExternalWritable := 'False'} : Int := 5;   // Minimum size parcel [mm] to set when no size is found
      ReactivationRequestDelay { ExternalAccessible := 'False'; ExternalVisible := 'False'; ExternalWritable := 'False'} : DInt := 10000;   // Delay distance before request to MergeGenerator to activate [mm]
      RunEmptyDistance : DInt := 10000;   // Distance the merge conveyor has to run before the induct starts after an EMstop [mm]
      SearchOnly { ExternalAccessible := 'False'; ExternalVisible := 'False'; ExternalWritable := 'False'} : Bool;   // 1 = The induct is not requesting a gap, only searching
      DistanceRunBeforeAutoRecovery : Int := 1;   // Distance the merge conevyor should run before Induct does an auto recovery request
      ParcelStopPositionAutoRecovery : Int;   // Position where parcel stops when Induct needs to auto recover
      RecoveryAdditionalGap : Int;   // Additional Gap during recovery  or first startup of Induct
      InductPositionWindow : Int := 10;   // Induct position window (tollerance) [cm]
      FlexGap { ExternalAccessible := 'False'; ExternalVisible := 'False'; ExternalWritable := 'False'} : Array[1..5] of "UDT_InductGapsize";
   END_STRUCT;

END_TYPE

DATA_BLOCK "DB_Time"
TITLE = DB_Time
{ S7_Optimized_Access := 'TRUE' }
AUTHOR : MHSE
FAMILY : GeneralSystemFunctions
VERSION : 3.0
NON_RETAIN
//Data block to store date and time data.
   VAR
      ActualTimeDTL {InstructionName := 'DTL'; LibVersion := '1.0'; ExternalAccessible := 'False'; ExternalVisible := 'False'; ExternalWritable := 'False'} : DTL;   // Actual date and time in DTL
      ActualTime { ExternalAccessible := 'False'; ExternalVisible := 'False'; ExternalWritable := 'False'} : String;   // Actual date and time in String
      Timestamp { ExternalAccessible := 'False'; ExternalVisible := 'False'; ExternalWritable := 'False'} : String[17];   // Actual date and time in String
      DaylightSaving { ExternalAccessible := 'False'; ExternalVisible := 'False'; ExternalWritable := 'False'} : Int;
   END_VAR


BEGIN

END_DATA_BLOCK

TYPE "UDT_InchingStatus"
VERSION : 0.1
   STRUCT
      Full { ExternalAccessible := 'False'; ExternalVisible := 'False'; ExternalWritable := 'False'} : Bool;   // Conveyor is full
      Active { ExternalAccessible := 'False'; ExternalVisible := 'False'; ExternalWritable := 'False'} : Bool;   // Inching is active
   END_STRUCT;

END_TYPE

TYPE "UDT_Destinations"
VERSION : 0.1
   STRUCT
      Destination : Array[0..5] of DInt;   // Destination code to compare to to go to position
   END_STRUCT;

END_TYPE

TYPE "UDT_GapOptimizationSystemConfiguration"
VERSION : 0.1
   STRUCT
      LengthConvA : Int;   // The length of conveyor A (mm)
      LengthConvB : Int;   // The length of conveyor B (mm)
      LengthConvC : Int;   // The length of conveyor C (mm)
      PosPECA1 : Int;   // The position of PEC from the beginning of conveyor A (mm)
      PosPECA2 : Int;   // The position of PEC from the end of the conveyor A (mm)
      PosPECB1 : Int;   // The position of PEC from the beginning of conveyor B (mm)
      PosPECB2 : Int;   // The position of PEC from the end of the conveyor B (mm)
      PosPECC1 : Int;   // The position of PEC from the beginning of conveyor C (mm)
      PosPECC2 : Int;   // The position of PEC from the end of the conveyor C (mm)
      InitialSpeed : Int;   // Initial speed of each conveyor (mm/s)
      Acceleration : Int;   // Acceleration (mm/s2)
      MaximumSpeed : Int;   // Maximum speed (mm/s)
      MinimumSpeed : Int;   // Minimum speed (mm/s)
      MarginLength : Int;   // Extra length margin for acceleration (mm)
      RequiredGap : Int;   // The required gap (mm)
      AllowedUpstreamGap : Int;   // Minimum upstream gap allowed to decelerate (mm)
      AllowedParcelLength : Int;   // The maximum length of a parcel allowed to accelerate or decelerate on one conveyor (mm)
      LengthSpaceBetweenConv : Int;   // The distance of free space between 2 conveyors (mm)
      PosPECBos : Int;   // The position of the PEC from the beginning of the conveyor (mm)
   END_STRUCT;

END_TYPE

TYPE "UDT_GapOptimizationSystemStatus"
VERSION : 0.1
   STRUCT
      Status : Int;   // Status number
   END_STRUCT;

END_TYPE

TYPE "UDT_GapOptimizationSystemInterface"
VERSION : 0.1
   STRUCT
      SpeedConvA : Int;   // Setpoint speed of conveyor A (mm/s)
      SpeedConvB : Int;   // Setpoint speed of conveyor B (mm/s)
      SpeedConvC : Int;   // Setpoint speed of conveyor C (mm/s)
   END_STRUCT;

END_TYPE

FUNCTION "FC_GOSCalculation" : Void
{ S7_Optimized_Access := 'TRUE' }
VERSION : 0.1
// ATTRIBUTES
// AUTO_NUMBER = True
// BLOCK_NUMBER = 21
// END_ATTRIBUTES
   VAR_INPUT
      ir_TravelDistanceCurrentParc : Real;   // Travel distance of the current parcel till the end of the conveyor (mm)
      ir_TravelDistanceUpstreamParc : Real;   // Travel distance of the upstream parcel till the end of the conveyor (mm)
      ir_InitialSpeed : Real;   // Initial speed of the VFD (mm/s)
      ir_Acceleration : Real;   // Maximum acceleration of the VFD (mm/s2)
      ir_MaxSpeed : Real;   // Maximum speed of the VFD (mm/s)
      ir_MinSpeed : Real;   // Minimum speed of hte VFD (mm/s)
      ii_ParcelGapDownstream : Int;   // Downstream gap of the current parcel to his next parcel (mm)
      ii_ParcelGapUpstream : Int;   // Upstream gap of the current parcel to his previous parcel (mm)
      ii_RequiredGap : Int;   // Required gap between the parcels (mm)
      ii_MarginGap : Int;   // Extra margin gap (mm)
      ii_AllowedUpstreamGap : Int;   // Maximum allowed gap upstream (mm)
      ix_ActionConv : Bool;   // ActionConv = True means that conveyor is running
   END_VAR

   VAR_OUTPUT
      qi_Speed : Int;   // Calculated speed (mm/s)
      qi_ParcelGapRecovered : Int;   // Gap recovered by acceleration or deceleration (mm)
      qx_Accelerate : Bool;   // Accelerate = True means that the action of acceleration is active
      qx_Decelerate : Bool;   // Decelerate = True means that the action of deceleration is active
      qi_TimeToChangeSpeed : LReal;   // Time for which the speed shoud be changed  [ms]
   END_VAR

   VAR_TEMP
      tr_NewTravelTime : Real;   // Calculated travel time (s)
      tr_Speed : Real;   // Calculated speed (mm/s)
      tr_RecoverdGapAccDec : Real;   // Gap that is recovered by acceleration and deceleration (mm)
      tr_RecoverdGapDecAcc : Real;   // Gap that is recovered by deceleration and acceleration (mm)
      tr_ParcelGapToBeRecovered : Real;   // Gap that has to be recovered (mm)
      tr_NewTravelDistance : Real;   // Calculated travel distance (mm)
      tr_AccDecTravelDistance : Real;   // Distance travelled by parcel when accelerated and decelerated (mm)
   END_VAR


BEGIN
	(*

	----------------------------------------------------------------------------------------
	28/01/2020  | 1.0       | R. Joosse     | first release TIA 15.1
	28/01/2020  | 2.0       | M. Singh      | Used Absolute value of input distances so as to have correct calculations in case of a UFO
	04/04/2023  | 4.0       | F.Baten       | 4.0 Release TIA 17.5
	*)

	REGION 1 Calculation speed for acceleration and deceleration
	    //Acceleration

	    IF ((#ii_ParcelGapDownstream > #ii_RequiredGap + #ii_MarginGap) AND (#ii_ParcelGapUpstream < #ii_RequiredGap) AND (#ii_ParcelGapUpstream <> 0))
	        OR (#ii_ParcelGapDownstream > #ii_RequiredGap + 100) //100mm is to be added to Config as "Additional Gap Downstream For Unconditional Acccelaeration"
	    THEN
	        #tr_ParcelGapToBeRecovered := #ii_ParcelGapDownstream - #ii_RequiredGap;
	        #qx_Accelerate := True;
	        #qx_Decelerate := FALSE;

	        IF #ix_ActionConv
	        THEN
	            IF ABS_REAL(IN := #ir_TravelDistanceUpstreamParc) <= ABS_REAL(IN := #ir_TravelDistanceCurrentParc)

	            THEN
	                #tr_NewTravelDistance := ABS_REAL(IN := #ir_TravelDistanceUpstreamParc); //   #tr_NewTravelDistance := #ir_TravelDistance_UpstreamParc;
	            ELSE
	                #tr_NewTravelDistance := ABS_REAL(IN := #ir_TravelDistanceCurrentParc); //    #tr_NewTravelDistance := #ir_TravelDistance_CurrentParc;
	            END_IF;

	            //Calculate speed  (v2 = u2 +2as)
	            #tr_Speed := SQRT((#ir_InitialSpeed * #ir_InitialSpeed) + (2.0 * #ir_Acceleration * ((#tr_NewTravelDistance / 2.0))));

	            // #tr_Speed := SQRT((#ir_InitialSpeed * #ir_InitialSpeed) + (2.0 * #ir_Acceleration * ((#tr_NewTravelDistance / 2.0) - 50)));
	            //Calculate travel time (v = u + at)
	            #tr_NewTravelTime := ((#tr_Speed - #ir_InitialSpeed) / #ir_Acceleration) * 2.0;

	            //Recovered gap by acceleration and deceleration in millimeters
	            #tr_RecoverdGapAccDec := #tr_NewTravelDistance - (#ir_InitialSpeed * #tr_NewTravelTime);

	            IF #tr_RecoverdGapAccDec <= #tr_ParcelGapToBeRecovered
	            THEN
	                #qi_ParcelGapRecovered := REAL_TO_INT(#tr_RecoverdGapAccDec);
	            ELSE
	                #tr_NewTravelDistance := #tr_NewTravelDistance - (#tr_RecoverdGapAccDec - #tr_ParcelGapToBeRecovered);

	                #tr_Speed := SQRT((#ir_InitialSpeed * #ir_InitialSpeed) + (2.0 * #ir_Acceleration * ((#tr_NewTravelDistance / 2.0))));

	                //   #tr_Speed := SQRT((#ir_InitialSpeed * #ir_InitialSpeed) + (2.0 * #ir_Acceleration * ((#tr_NewTravelDistance / 2.0) - 50)));

	                //Calculate travel time (v = u + at)
	                #tr_NewTravelTime := ((#tr_Speed - #ir_InitialSpeed) / #ir_Acceleration) * 2.0;

	                #qi_ParcelGapRecovered := REAL_TO_INT(#tr_NewTravelDistance - (#ir_InitialSpeed * #tr_NewTravelTime));
	            END_IF;
	        END_IF;

	        //Deceleration
	    ELSIF (#ii_ParcelGapDownstream < #ii_RequiredGap) AND #ii_ParcelGapDownstream > 0 AND
	        ((#ii_ParcelGapUpstream > #ii_AllowedUpstreamGap) OR (#ii_ParcelGapUpstream = 0))

	    THEN
	        #tr_ParcelGapToBeRecovered := #ii_RequiredGap - #ii_ParcelGapDownstream;
	        #qx_Accelerate := FALSE;
	        #qx_Decelerate := True;

	        IF #ix_ActionConv
	        THEN
	            IF ABS_REAL(IN := #ir_TravelDistanceUpstreamParc) <= ABS_REAL(IN := #ir_TravelDistanceCurrentParc) AND
	                (ABS_REAL(IN := #ir_TravelDistanceUpstreamParc) > 150.0)
	            THEN
	                #tr_NewTravelDistance := ABS_REAL(IN := #ir_TravelDistanceUpstreamParc);
	            ELSE
	                #tr_NewTravelDistance := ABS_REAL(IN := #ir_TravelDistanceCurrentParc);
	            END_IF;

	            //Calculate speed used v2 = (u2 -2as)
	            #tr_Speed := SQRT((#ir_InitialSpeed * #ir_InitialSpeed) - ((2.0 * #ir_Acceleration * (#tr_NewTravelDistance / 2.0))));

	            //Calculate travel time v= u + at
	            #tr_NewTravelTime := ((#ir_InitialSpeed - #tr_Speed) / #ir_Acceleration) * 2.0;

	            //Recovered gap by acceleration and deceleration in millimeters
	            #tr_RecoverdGapDecAcc := (#ir_InitialSpeed * #tr_NewTravelTime) - #tr_NewTravelDistance;

	            IF #tr_RecoverdGapDecAcc <= #tr_ParcelGapToBeRecovered
	            THEN
	                #qi_ParcelGapRecovered := REAL_TO_INT(#tr_RecoverdGapDecAcc);
	            ELSE
	                #tr_NewTravelDistance := #tr_NewTravelDistance - (#tr_RecoverdGapDecAcc - #tr_ParcelGapToBeRecovered);

	                //Calculate speed used v2 = (u2 -2as)
	                #tr_Speed := SQRT((#ir_InitialSpeed * #ir_InitialSpeed) - ((2.0 * #ir_Acceleration * (#tr_NewTravelDistance / 2.0))));

	                //Calculate travel time v= u + at
	                #tr_NewTravelTime := ((#ir_InitialSpeed - #tr_Speed) / #ir_Acceleration) * 2.0;

	                //Recovered gap by acceleration and deceleration in millimeters
	                #tr_RecoverdGapDecAcc := (#ir_InitialSpeed * #tr_NewTravelTime) - #tr_NewTravelDistance;

	                #qi_ParcelGapRecovered := REAL_TO_INT(#tr_RecoverdGapDecAcc);

	            END_IF;
	        END_IF;

	    ELSE
	        //Initial speed
	        #tr_Speed := #ir_InitialSpeed;
	        #qx_Accelerate := FALSE;
	        #qx_Decelerate := FALSE;
	    END_IF;
	END_REGION

	REGION 2 Write calculated speed on the output
	    #qi_TimeToChangeSpeed := REAL_TO_LREAL(IN := #tr_NewTravelTime * 1000 / 2);

	    IF #tr_Speed > #ir_InitialSpeed
	    THEN
	        #qi_Speed := REAL_TO_INT(#ir_MaxSpeed);
	    ELSIF #tr_Speed < #ir_InitialSpeed
	    THEN
	        #qi_Speed := REAL_TO_INT(#ir_MinSpeed);
	    END_IF;
	END_REGION


END_FUNCTION

TYPE "UDT_Merge"
VERSION : 0.1
   STRUCT
      LastUsed : Int;   // Last used FIFO entry
      MaxNumberofEntries : Int;   // Maximum number of FIFO entries
      Remove { ExternalAccessible := 'False'; ExternalVisible := 'False'; ExternalWritable := 'False'} : Bool;   // An entry was removed by an induct
      GenerationInactive { ExternalAccessible := 'False'; ExternalVisible := 'False'; ExternalWritable := 'False'} : Bool;   // Generation is inactive (not generating and handling requests)
      ReactivateReq { ExternalAccessible := 'False'; ExternalVisible := 'False'; ExternalWritable := 'False'} : Bool;   // Request to activate generation from an induct
      FIFO : Array[0..10] of "UDT_FIFOInductInfo";   // FIFO structure for induct requests
      TrackingPointerForInduct { S7_SetPoint := 'True'} : Array[1..10] of Int;   // Tracking the request for the induct
      RequestInFIFO { S7_SetPoint := 'True'} : Array[1..10] of Bool;   // Request is in FIFO handshake
   END_STRUCT;

END_TYPE

DATA_BLOCK "DB_GOSLog"
{ S7_Optimized_Access := 'TRUE' }
VERSION : 0.1
NON_RETAIN
   VAR
      DB_GOSLog { ExternalAccessible := 'False'; ExternalVisible := 'False'; ExternalWritable := 'False'; S7_SetPoint := 'False'} : Array[0..100] of "UDT_GOSLog";
   END_VAR


BEGIN

END_DATA_BLOCK

TYPE "UDT_ConveyorPanelStatus"
TITLE = Cabinet MCP Status
VERSION : 0.1
   STRUCT
      CBFeedbackError { ExternalAccessible := 'False'; ExternalVisible := 'False'; ExternalWritable := 'False'} : Bool;   // Circuit feedback error
      MainSwitchOff { ExternalAccessible := 'False'; ExternalVisible := 'False'; ExternalWritable := 'False'} : Bool;   // Main switch tripped
   END_STRUCT;

END_TYPE

TYPE "UDT_ConveyorPanelStatistics"
TITLE = Cabinet MCP Statistics
VERSION : 0.1
   STRUCT
      CBFeedbackError : "UDT_EventStatistic";   // Circuit breaker feedback error
      MainSwitchOff : "UDT_EventStatistic";   // Main switch fault statistics
   END_STRUCT;

END_TYPE

TYPE "UDT_ControlPowerGroupStatus"
VERSION : 0.1
   STRUCT
      Status : Int;   // Status number
      Specific : Struct
         Fail_PowerSupply_1 { ExternalAccessible := 'False'; ExternalVisible := 'False'; ExternalWritable := 'False'} : Bool;   // Power supply 1 fail
         Fail_PowerSupply_2 { ExternalAccessible := 'False'; ExternalVisible := 'False'; ExternalWritable := 'False'} : Bool;   // Power supply 2 fail
         Fail_PowerSupply_3 { ExternalAccessible := 'False'; ExternalVisible := 'False'; ExternalWritable := 'False'} : Bool;   // Power supply 3 fail
         Fail_PowerSupply_4 { ExternalAccessible := 'False'; ExternalVisible := 'False'; ExternalWritable := 'False'} : Bool;   // Power supply 4 fail
         Fail_PowerSupply_5 { ExternalAccessible := 'False'; ExternalVisible := 'False'; ExternalWritable := 'False'} : Bool;   // Power supply 5 fail
         Fail_PowerSupply_6 { ExternalAccessible := 'False'; ExternalVisible := 'False'; ExternalWritable := 'False'} : Bool;   // Power supply 6 fail
         Fail_PowerSupply_7 { ExternalAccessible := 'False'; ExternalVisible := 'False'; ExternalWritable := 'False'} : Bool;   // Power supply 7 fail
         Fail_PowerSupply_8 { ExternalAccessible := 'False'; ExternalVisible := 'False'; ExternalWritable := 'False'} : Bool;   // Power supply 8 fail
         Fail_PowerSupply_9 { ExternalAccessible := 'False'; ExternalVisible := 'False'; ExternalWritable := 'False'} : Bool;   // Power supply 9 fail
         Fail_PowerSupply_10 { ExternalAccessible := 'False'; ExternalVisible := 'False'; ExternalWritable := 'False'} : Bool;   // Power supply 10 fail
         PowerSuppliesWarning { ExternalAccessible := 'False'; ExternalVisible := 'False'; ExternalWritable := 'False'} : Bool;   // Power supplies warning
         PowerSuppliesError { ExternalAccessible := 'False'; ExternalVisible := 'False'; ExternalWritable := 'False'} : Bool;   // Power supplies error
      END_STRUCT;
   END_STRUCT;

END_TYPE

TYPE "UDT_ControlPowerGroupStatistics"
VERSION : 0.1
   STRUCT
      PowerSupplyGroupWarnning : "UDT_EventStatistic";   // Warning Power Supply Group Statistics
      PowerSupplyGroupError : "UDT_EventStatistic";   // Error Power Supply Group Statistics
   END_STRUCT;

END_TYPE

TYPE "UDT_AirPressureSwitchStatus"
VERSION : 0.1
   STRUCT
      Status : Int;   // Status number
      Specific : Struct   // Equipment specific warnings and errors
         AirPressureOK : Bool;   // Air pressure switch is okay
      END_STRUCT;
   END_STRUCT;

END_TYPE

TYPE "UDT_TPManualControlButtons"
TITLE = UDT_TPManualControlButtons
VERSION : 0.1
//User defined structure to communicate buttons to and from the Touch buttons
   STRUCT
      ManualMode : Bool;
      ManualStart : Bool;
      ManualStop : Bool;
      ManualFullSpeed : Bool;
      ManualLowSpeed : Bool;
      ManualJog : Bool;
      ManualReverse : Bool;
   END_STRUCT;

END_TYPE

TYPE "UDT_AixPlcFull4McoStatus"
VERSION : 0.1
   STRUCT
      StatusMotor1 { S7_SetPoint := 'False'} : "UDT_AixControllerStatus";
      StatusMotor2 : "UDT_AixControllerStatus";
      StatusMotor3 : "UDT_AixControllerStatus";
      StatusMotor4 : "UDT_AixControllerStatus";
      StatusMotor5 : "UDT_AixControllerStatus";
      StatusMotor6 : "UDT_AixControllerStatus";
      StatusMotor7 : "UDT_AixControllerStatus";
      StatusMotor8 : "UDT_AixControllerStatus";
   END_STRUCT;

END_TYPE

FUNCTION "FC_StringToTime" : Void
TITLE = FC_StringToTime
{ S7_Optimized_Access := 'TRUE' }
AUTHOR : MHSE
FAMILY : GeneralSystemFunctions
VERSION : 3.0
// ATTRIBUTES
// AUTO_NUMBER = True
// BLOCK_NUMBER = 27
// END_ATTRIBUTES
//Function to convert date in string format to the DTL.
   VAR_INPUT
      is_StringTime : String;   // Input string with date
   END_VAR

   VAR_OUTPUT
      qt_Date {InstructionName := 'DTL'; LibVersion := '1.0'} : DTL;   // Output Date in DTL
   END_VAR

   VAR_TEMP
      ts_DateInt : Struct   // Temp partial date in integer
         Year : UInt;
         Month : USInt;
         Day : USInt;
         Hour : USInt;
         Minute : USInt;
         Second : USInt;
         Millisecond : UDInt;
      END_STRUCT;
      ts_DateString : Struct   // Temp partial date in string
         Hour : String[2];
         Minute : String[2];
         Second : String[2];
         Millisecond : String[3];
      END_STRUCT;
   END_VAR

   VAR CONSTANT
      ci_StringLength2 : Int := 2;   // Length of the part of the string
      ci_StringLength3 : Int := 3;   // Length of the part of the string
      ci_StringPosition1 : Int := 1;   // Position of the first caracter inside the string
      ci_StringPosition4 : Int := 4;   // Position of the first caracter inside the string
      ci_StringPosition7 : Int := 7;   // Position of the first caracter inside the string
      ci_StringPosition10 : Int := 10;   // Position of the first caracter inside the string
      cw_FormatZero : Word := 0;   // Simple value format
      Ci_Year : UInt := 1970;   // Fixed year 1970, start value dtl
      ci_Month : USInt := 1;   // Fixed month 1, start value dtl
      ci_Day : USInt := 1;   // Fixed day 1, start value dtl
   END_VAR


BEGIN
	(*
	----------------------------------------------------------------------------------------

	Version history:
	Date        | Version   | Author        | Remark
	----------------------------------------------------------------------------------------
	24/05/2019  | 0.1       | K.Pokorski    | first release MHS TIA 15.1
	26/06/2019  | 0.2       | M.Kurpiers    | Change in region 1 P:=3 -> P:=4
	24/07/2019  | 2.0       | L.Klar        | 2.0 MHS library release TIA 15.1
	26/07/2019  | 2.1       | M.Kurpiers    | Comments adjusted
	12/11/2019  | 3.0       | P.Majka       | 3.0 MHS library release TIA 15.1
	16/02/2023  | 3.1       | F.Baten       | Added constants
	21/02/2023  | 4.0       | F.Baten       | 4.0 Release TIA 17.5
	*)

	REGION 1 - Separation different part of the date

	    // Separation different part of the date from the data string and saving it to the structure
	    #ts_DateString.Hour := MID(IN := #is_StringTime,
	                               L := #ci_StringLength2,
	                               P := #ci_StringPosition1);               // Separating an hour from the date string
	    #ts_DateString.Minute := MID(IN := #is_StringTime,
	                                 L := #ci_StringLength2,
	                                 P := #ci_StringPosition4);             // Separating a minute from the date string
	    #ts_DateString.Second := MID(IN := #is_StringTime,
	                                 L := #ci_StringLength2,
	                                 P := #ci_StringPosition7);             // Separating a second from the date string
	    #ts_DateString.Millisecond := MID(IN := #is_StringTime,
	                                      L := #ci_StringLength3,
	                                      P := #ci_StringPosition10);       // Separating a millisecond from the date string

	END_REGION

	REGION 2 - Conversion string to integer

	    STRG_VAL(IN := #ts_DateString.Hour,                         // Conversion a hour from string
	             FORMAT := #cw_FormatZero,                          // Simple value format
	             P := INT_TO_UINT(#ci_StringPosition1),             // First position in string
	             OUT => #ts_DateInt.Hour);                          // Integer temporary variable
	    // Conversion a minute from string
	    STRG_VAL(IN := #ts_DateString.Minute,
	             FORMAT := #cw_FormatZero,
	             P := INT_TO_UINT(#ci_StringPosition1),
	             OUT => #ts_DateInt.Minute);
	    // Conversion a second from string
	    STRG_VAL(IN := #ts_DateString.Second,
	             FORMAT := #cw_FormatZero,
	             P := INT_TO_UINT(#ci_StringPosition1),
	             OUT => #ts_DateInt.Second);
	    // Conversion a milisecond from string
	    STRG_VAL(IN := #ts_DateString.Millisecond,
	             FORMAT := #cw_FormatZero,
	             P := INT_TO_UINT(#ci_StringPosition1),
	             OUT => #ts_DateInt.Millisecond);

	END_REGION

	REGION 3 - Combine integer to "DTL" data type and setting output

	    // Move parts of the date to the DTL output structure
	    #qt_Date.YEAR := #Ci_Year;
	    #qt_Date.MONTH := #ci_Month;
	    #qt_Date.DAY := #ci_Day;
	    #qt_Date.HOUR := #ts_DateInt.Hour;
	    #qt_Date.MINUTE := #ts_DateInt.Minute;
	    #qt_Date.SECOND := #ts_DateInt.Second;
	    #qt_Date.NANOSECOND := #ts_DateInt.Millisecond * 1000000;

	END_REGION
END_FUNCTION

TYPE "UDT_PNCoupler_Interface"
TITLE = Interface signals between PN Coupler
VERSION : 0.1
   STRUCT
      DownstreamDisplacement : Int;   // Displacement from downstream [cm]
      RTS : Bool;   // Conveyor ready to send
      RTR : Bool;   // Conveyor ready to receive
      TIP : Bool;   // Transfer in progress
      ResetEnergySave : Bool;   // Reset energy save mode
      CascadeStartUp : Bool;   // Cascade startup
   END_STRUCT;

END_TYPE

TYPE "UDT_EncoderStatus"
VERSION : 0.1
   STRUCT
      Fault { ExternalAccessible := 'False'; ExternalVisible := 'False'; ExternalWritable := 'False'} : Bool;
   END_STRUCT;

END_TYPE

TYPE "UDT_MergeGeneratorConfig"
TITLE = UDT_MergeGeneratorConfig
VERSION : 0.1
//V 3.1
   STRUCT
      GenerationPoint : Int;   // Position on tracking where is written [mm]
      NumberInducts : Int;   // Number of induct belts conected to the merge belt.
      GapHeadToHead : Int;   // Length of the fixed gap (cm)
      ChangeWindowModeDistance : DInt := 60000;   // Distance to Deactivate window generation (mm)
      ModeSelection : Int;   // 0= standard, 1 = no empty window
      DelayDistance : Int;   // Delay in looking for next window for the same induct
   END_STRUCT;

END_TYPE

FUNCTION_BLOCK "FB_PECD"
TITLE = FB_PEC
{ S7_Optimized_Access := 'TRUE' }
AUTHOR : MHSE
FAMILY : Conveyor
VERSION : 3.0
// ATTRIBUTES
// AUTO_NUMBER = True
// BLOCK_NUMBER = 22
// END_ATTRIBUTES
   VAR_INPUT
      iUDT_PECConfiguration { ExternalAccessible := 'False'; ExternalVisible := 'False'; ExternalWritable := 'False'} : "UDT_PECDConfiguration";   // PEC configuration structure
      ix_PEC { ExternalAccessible := 'False'; ExternalVisible := 'False'; ExternalWritable := 'False'} : Bool;   // Signal of the PEC
   END_VAR

   VAR_OUTPUT
      qUDT_HMIStatus { ExternalAccessible := 'False'; ExternalVisible := 'False'; ExternalWritable := 'False'} : "UDT_PECStatus";   // Status structure
      qx_PECFiltered { ExternalAccessible := 'False'; ExternalVisible := 'False'; ExternalWritable := 'False'} : Bool;   // PEC Filtered
   END_VAR

   VAR_IN_OUT
      iqUDT_ConveyorInterface : "UDT_ConveyorInterface";   // Interface structure
      iqUDT_PECStatistics : "UDT_PECStatistics";   // Statistics structure
   END_VAR

   VAR
      s_Status { ExternalAccessible := 'False'; ExternalVisible := 'False'; ExternalWritable := 'False'; S7_SetPoint := 'False'} : "UDT_PECStatus";   // Status structure
      s_StatusOld { ExternalAccessible := 'False'; ExternalVisible := 'False'; ExternalWritable := 'False'; S7_SetPoint := 'False'} : "UDT_PECStatus";   // Auxiliary status structure
      PEC_OnOffDelay { ExternalAccessible := 'False'; ExternalVisible := 'False'; ExternalWritable := 'False'; S7_SetPoint := 'False'} : "FB_OnOffDelayDistance";   // Filtering end of section photo eye signal
      R_TRIG_PECJam {InstructionName := 'R_TRIG'; LibVersion := '1.0'; ExternalAccessible := 'False'; ExternalVisible := 'False'; ExternalWritable := 'False'; S7_SetPoint := 'False'} : R_TRIG;   // Rising edge trigger PEC jam
      sx_Enable { ExternalAccessible := 'False'; ExternalVisible := 'False'; ExternalWritable := 'False'} : Bool;   // Enable
   END_VAR
   VAR RETAIN
      si_AuxJamDisplacement { ExternalAccessible := 'False'; ExternalVisible := 'False'; ExternalWritable := 'False'} : Int;   // Auxiliary variable to calculate displacement when PEC is blocked
   END_VAR
   VAR
      sx_PECFiltered { ExternalAccessible := 'False'; ExternalVisible := 'False'; ExternalWritable := 'False'} : Bool;   // Photo eye filtered
   END_VAR


BEGIN
	(*
	----------------------------------------------------------------------------------------

	Version history:
	Date        | Version   | Author        | Remark
	----------------------------------------------------------------------------------------
	 16/04/2023 | 1.0       | F.Baten       | Adapt from PEC timer based
	 03/05/2023 | 4.0       | F.Baten       | 4.0 Release TIA 17.5
	*)

	REGION 1 - Triggers

	    // Rising edge PEC Jam
	    #R_TRIG_PECJam(CLK := #s_Status.Jam);

	END_REGION

	REGION 2 - Active function

	    // To activate the jam monitoring the jam displacement limit  must be configured up to zero.
	    #sx_Enable := #iUDT_PECConfiguration.JamDisplacementLimit > 0;

	END_REGION

	REGION 3 - Reset errors

	    // Jam error is reset when reset bit is active and jam error is active and is connfigured alllow reset jam with PEC blocked or photo eye is not active
	    IF #iqUDT_ConveyorInterface.InternalErrorReset
	        AND (#iUDT_PECConfiguration.ResetWithPECBlocked
	        OR (NOT #iUDT_PECConfiguration.ResetWithPECBlocked
	        AND #sx_PECFiltered))
	        AND #s_Status.Jam
	    THEN

	        #si_AuxJamDisplacement := 0;
	        #s_Status.Jam := FALSE;

	    END_IF;

	END_REGION

	REGION 4 - Photo eye filters

	    // End of section photo eye signal filter measurement
	    #PEC_OnOffDelay(ii_Displacement := #iqUDT_ConveyorInterface.Displacement,
	                    idi_OnDelayDistance := #iUDT_PECConfiguration.OnDelayDistance,
	                    idi_OffDelayDistance := #iUDT_PECConfiguration.OffDelayDistance,
	                    ix_SignalToDelay := #ix_PEC,
	                    ix_Enable := TRUE,
	                    qx_DelayedSignal => #sx_PECFiltered);

	    // Write the current status of the photo eye
	    #s_Status.PEC := #sx_PECFiltered;
	    #qx_PECFiltered := #sx_PECFiltered;

	END_REGION

	REGION 5 - Jam detection

	    IF NOT #sx_PECFiltered                                             // Photo eye blocked
	        AND #sx_Enable                                                  // Active of checking the PEC jam
	    THEN

	        #si_AuxJamDisplacement += ABS(#iqUDT_ConveyorInterface.Displacement);

	    ELSE

	        #si_AuxJamDisplacement := 0;

	    END_IF;

	    // Compare jam auxiliary counter with displacement jam configured
	    IF #si_AuxJamDisplacement > #iUDT_PECConfiguration.JamDisplacementLimit
	    THEN

	        #s_Status.Jam := TRUE;

	    END_IF;

	END_REGION

	REGION 6 - Statistics

	    // Statistics Jam PEC
	    IF #s_Status.Jam                                                    // PEC jam error active
	        OR #iqUDT_ConveyorInterface.ResetStatistics                    // Reset statistics
	    THEN

	        "FC_Statistics"(ix_Reset := #iqUDT_ConveyorInterface.ResetStatistics,
	                        ix_Activate := #s_Status.Jam,
	                        ix_RTrigActivate := #R_TRIG_PECJam.Q,
	                        iqUDT_Statistics := #iqUDT_PECStatistics.Jam);

	    END_IF;

	END_REGION

	REGION 7 - Internal PEC error

	    IF #s_Status.Jam
	    THEN

	        #iqUDT_ConveyorInterface.InternalErrorPEC := TRUE;

	    END_IF;

	END_REGION


	REGION 8 - Status

	    // Status update on change
	    IF #s_StatusOld <> #s_Status
	    THEN

	        #qUDT_HMIStatus := #s_Status;
	        #s_StatusOld := #s_Status;

	    END_IF;

	END_REGION
END_FUNCTION_BLOCK

TYPE "UDT_PECDUpdateConfiguration"
TITLE = UDT_PECConfiguration
VERSION : 0.1
//User-defined structure of PEC parameters.
   STRUCT
      OnDelayDistance : DInt;   // Photo eye distance on delay [cm]
      OffDelayDistance : DInt;   // Photo eye distance off delay [cm]
      Distance : DInt;   // Distance between photo eye and the end of conveyor [mm]
      JamDisplacementLimit : Int;   // Limit displacement with PEC blocked o detect jam [cm]
      SearchWindowFwd : Int;   // Search window in forward direction [cm]
      SearchWindowRvs : Int;   // Search window in reverse direction [cm]
      GINRangeStart : Int;   // GIN range start value
      GINRangeEnd : Int;   // GIN range end value
      NrOfTeachParcels : Int;   // Number of parcels to teach
      DefaultGIN : Int := 1;   // Default GIN record
      MaxLost : Int;   // Maximum number of lost parcels in a row
      ParcelLengthFilter : Bool := TRUE;   // Parcel length filter
      ResetWithPECBlocked { ExternalAccessible := 'False'; ExternalVisible := 'False'; ExternalWritable := 'False'} : Bool;   // When 'True' Allow reset system after jam with PEC blocked
      GenerationPoint { ExternalAccessible := 'False'; ExternalVisible := 'False'; ExternalWritable := 'False'} : Bool;   // Generation point
      NegativeGINDelete { ExternalAccessible := 'False'; ExternalVisible := 'False'; ExternalWritable := 'False'} : Bool;   // True when negative GIN has to be deleted
      ParcelLengthMeasurement { ExternalAccessible := 'False'; ExternalVisible := 'False'; ExternalWritable := 'False'} : Bool;   // Parcel length measurement
      GapLengthMeasurement { ExternalAccessible := 'False'; ExternalVisible := 'False'; ExternalWritable := 'False'} : Bool;   // Gap length measurement
   END_STRUCT;

END_TYPE

TYPE "UDT_WE01Status"
VERSION : 0.1
   STRUCT
      Status : Int;   // Status number
      Specific : Struct
         WeighingScaleFault { ExternalAccessible := 'False'; ExternalVisible := 'False'; ExternalWritable := 'False'} : Bool;   // Weighing Scale unit in Fault state
      END_STRUCT;
   END_STRUCT;

END_TYPE

TYPE "UDT_VSUConfiguration"
TITLE = UDT_VSUConfig
VERSION : 0.1
//User-defined structure of VSU parameters.
   STRUCT
      PEC_EoSTimeOnDelay { ExternalAccessible := 'False'; ExternalVisible := 'False'; ExternalWritable := 'False'} : UDInt;   // Photo eye EOS time on delay [ms]
      PEC_EoSTimeOffDelay { ExternalAccessible := 'False'; ExternalVisible := 'False'; ExternalWritable := 'False'} : UDInt;   // Photo eye EOS time off delay [ms]
      PEC_OutTimeOnDelay { ExternalAccessible := 'False'; ExternalVisible := 'False'; ExternalWritable := 'False'} : UDInt;   // Photo eye outfeed time on delay [ms]
      PEC_OutTimeOffDelay { ExternalAccessible := 'False'; ExternalVisible := 'False'; ExternalWritable := 'False'} : UDInt;   // Photo eye outfeed time off delay [ms]
      PEC_JamTimeOnDelay { ExternalAccessible := 'False'; ExternalVisible := 'False'; ExternalWritable := 'False'} : UDInt;   // Photo eye jam time on delay [ms]
      PEC_JamTimeOffDelay { ExternalAccessible := 'False'; ExternalVisible := 'False'; ExternalWritable := 'False'} : UDInt;   // Photo eye jam time off delay [ms]
      JogNoHornTime { ExternalAccessible := 'False'; ExternalVisible := 'False'; ExternalWritable := 'False'} : UDInt := 1000;   // Time within jog buttons can be pressed without new startup indication
      SwitchingTime { ExternalAccessible := 'False'; ExternalVisible := 'False'; ExternalWritable := 'False'} : UInt := 950;   // Time it takes to go from one position to the next [ms]
      DefaultPosition { ExternalAccessible := 'False'; ExternalVisible := 'False'; ExternalWritable := 'False'} : Int := 2;   // Default position number (1= up or 2= down) , If left 0 the block will go to 1
      HeadToHead { ExternalAccessible := 'False'; ExternalVisible := 'False'; ExternalWritable := 'False'} : Int := 120;   // Head to head distance to downstream conveyor (upper and lower) [cm]
      Gap { ExternalAccessible := 'False'; ExternalVisible := 'False'; ExternalWritable := 'False'} : Int := 60;   // Gap to downstream conveyor (upper and lower) [cm]
      JamDisplacementLimit { ExternalAccessible := 'False'; ExternalVisible := 'False'; ExternalWritable := 'False'} : Int := 100;   // Limit displacement with PEC blocked to detect jam [cm]
      SecurityChecked { ExternalAccessible := 'False'; ExternalVisible := 'False'; ExternalWritable := 'False'} : Bool;   // If true, then in semiautomatic stop the parcel for reject (if the VSU is not directed to reject)
   END_STRUCT;

END_TYPE

TYPE "UDT_VSUStatus"
TITLE = UDT_VSUStatus
VERSION : 0.1
//User-defined structure of FB_VerticalSwitch function block status.
   STRUCT
      Status : Int;   // Status number
      Specific : Struct   // Equipment specific warnings and errors
         ReferencedError { ExternalAccessible := 'False'; ExternalVisible := 'False'; ExternalWritable := 'False'} : Bool;   // VFD is not referenced
         UpperSwitchArea_Err { ExternalAccessible := 'False'; ExternalVisible := 'False'; ExternalWritable := 'False'} : Bool;   // Upper switching area PEC was activated when moving
         LowerSwitchArea_Err { ExternalAccessible := 'False'; ExternalVisible := 'False'; ExternalWritable := 'False'} : Bool;   // Lower switching area PEC was activated when moving
         UpperEntranceJam_Err { ExternalAccessible := 'False'; ExternalVisible := 'False'; ExternalWritable := 'False'} : Bool;   // Upper outfeed conveyor entrance PEC was blocked too long
         LowerEntranceJam_Err { ExternalAccessible := 'False'; ExternalVisible := 'False'; ExternalWritable := 'False'} : Bool;   // Lower outfeed conveyor entrance PEC was blocked too long
         Direction_Err { ExternalAccessible := 'False'; ExternalVisible := 'False'; ExternalWritable := 'False'} : Bool;   // Parcel should be rejected (in semi-automatic and security mode).
         Keyswitch_WRN { ExternalAccessible := 'False'; ExternalVisible := 'False'; ExternalWritable := 'False'} : Bool;   // Keyswitch is in '0' position
         UpperPosition { ExternalAccessible := 'False'; ExternalVisible := 'False'; ExternalWritable := 'False'} : Bool;   // Upper position reached
         LowerPosition { ExternalAccessible := 'False'; ExternalVisible := 'False'; ExternalWritable := 'False'} : Bool;   // Lower position reached
      END_STRUCT;
   END_STRUCT;

END_TYPE

TYPE "UDT_VSUCommand"
TITLE = UDT_VSUCommand
VERSION : 0.1
//User-defined structure of VSU commands.
   STRUCT
      SemiAutomaticMode { ExternalAccessible := 'False'; ExternalVisible := 'False'; ExternalWritable := 'False'} : Bool;   // Semiautomatic mode command from HMI
      ManualMode { ExternalAccessible := 'False'; ExternalVisible := 'False'; ExternalWritable := 'False'} : Bool;   // Manual mode command from HMI
      CommandUp { ExternalAccessible := 'False'; ExternalVisible := 'False'; ExternalWritable := 'False'} : Bool;   // Command from HMI to go to upper position in semiautomatic or manual mode
      CommandDown { ExternalAccessible := 'False'; ExternalVisible := 'False'; ExternalWritable := 'False'} : Bool;   // Command from HMI to go to lower position in semiautomatic or manual mode
      JogUp { ExternalAccessible := 'False'; ExternalVisible := 'False'; ExternalWritable := 'False'} : Bool;   // Command from HMI to Jog upwards
      JogDown { ExternalAccessible := 'False'; ExternalVisible := 'False'; ExternalWritable := 'False'} : Bool;   // Command from HMI to Jog downwards
      ReferenceRun { ExternalAccessible := 'False'; ExternalVisible := 'False'; ExternalWritable := 'False'} : Bool;   // Command from HMI to reference drive
   END_STRUCT;

END_TYPE

TYPE "UDT_VSUStatistics"
TITLE = UDT_VSUStatistics
VERSION : 0.1
//User-defined structure of FB_VerticalSwitch function block statistics.
   STRUCT
      UpTime { ExternalAccessible := 'False'; ExternalVisible := 'False'; ExternalWritable := 'False'} : "UDT_EventStatistic";   // VSU up time
      DownTime : "UDT_EventStatistic";   // VSU down time
      UpperSwitchArea_Error : "UDT_EventStatistic";   // Error statistics for VSU
      LowerSwitchArea_Error : "UDT_EventStatistic";   // Error statistics for VSU
      UpperEntranceJam_Error : "UDT_EventStatistic";   // Error statistics for VSU
      LowerEntranceJam_Error : "UDT_EventStatistic";   // Error statistics for VSU
      Direction_Error : "UDT_EventStatistic";   // Error statistics for VSU
   END_STRUCT;

END_TYPE

TYPE "UDT_VfdSiemensPI"
TITLE = UDT_VFD_Siemens_PI
VERSION : 0.1
//User-defined structure of VFD Siemens input telegram.
   STRUCT
      ZSW_1 : Struct   // Status Word Interconnection 1
         SpareBit8 { ExternalAccessible := 'False'; ExternalVisible := 'False'; ExternalWritable := 'False'} : Bool;   // Spare bit 8
         MasterControlRequested { ExternalAccessible := 'False'; ExternalVisible := 'False'; ExternalWritable := 'False'} : Bool;   // 1 = Master_control_requested (The automation system is requested to accept the inverter control) p 2080[9] = r0899.9
         SafetyTestRequired { ExternalAccessible := 'False'; ExternalVisible := 'False'; ExternalWritable := 'False'} : Bool;   // Only applicable in G120 with safety motion monitoring
         SpareBit11 { ExternalAccessible := 'False'; ExternalVisible := 'False'; ExternalWritable := 'False'} : Bool;   // Spare bit 11
         HoldingBrakeOpen { ExternalAccessible := 'False'; ExternalVisible := 'False'; ExternalWritable := 'False'} : Bool;   // 1 = Holding brake open (Signal open and close a motor holding brake) p 2080[12] = r 0899.12
         AlarmMotorOvertemp { ExternalAccessible := 'False'; ExternalVisible := 'False'; ExternalWritable := 'False'} : Bool;   // 0 = Alarm, motor overtemperature p2080[13] = r 2135.14
         MotorRotatesClockwise { ExternalAccessible := 'False'; ExternalVisible := 'False'; ExternalWritable := 'False'} : Bool;   // 1 = Motor rotates clockwise (Internal inverter actual value > 0), 0 = Motor rotates counterclockwise (Invertal inverter actual value < 0) p 2080[14] = 2197.3
         AlarmInverterThermalOverload { ExternalAccessible := 'False'; ExternalVisible := 'False'; ExternalWritable := 'False'} : Bool;   // 0 = Alarm, inverter thermal overload p 2080[15] = r0836.0 / r2135.15
         ReadyToStart { ExternalAccessible := 'False'; ExternalVisible := 'False'; ExternalWritable := 'False'} : Bool;   // 1 = Ready_to_start (Power supply switched in; electronics initialized; pulses locked) p 2080[0] = r 0899.0
         Ready { ExternalAccessible := 'False'; ExternalVisible := 'False'; ExternalWritable := 'False'} : Bool;   // 1 = Ready (Motor is switched on (ON/OFF1 = 1), no fault is active. With the command "Enable operation" (STW1.3), the inverterswitches on the motor) p 2080[1] = r 0899.1
         OperationEnabled { ExternalAccessible := 'False'; ExternalVisible := 'False'; ExternalWritable := 'False'} : Bool;   // 1 = Operation enabled (Motor follows setpoint. See control word 1 bit 3) p 2080[2] = r 0899.2
         FaultActive { ExternalAccessible := 'False'; ExternalVisible := 'False'; ExternalWritable := 'False'} : Bool;   // 1 = Fault_active (The inverter has a fault. Acknowledge fault using STW1.7) p 2080[3] = r 2139.3
         OFF2Inactive { ExternalAccessible := 'False'; ExternalVisible := 'False'; ExternalWritable := 'False'} : Bool;   // 1 = OFF2_inactive (Coast down to standstill is not active) p 2080[4] = r 0899.4
         OFF3Inactive { ExternalAccessible := 'False'; ExternalVisible := 'False'; ExternalWritable := 'False'} : Bool;   // 1 = OFF3_inactive (Quick stop is not active) p 2080[5] = r 0899.5
         SpareBit6 { ExternalAccessible := 'False'; ExternalVisible := 'False'; ExternalWritable := 'False'} : Bool;   // Spare bit 6
         AlarmActive { ExternalAccessible := 'False'; ExternalVisible := 'False'; ExternalWritable := 'False'} : Bool;   // 1 = Alarm_active (Motor remains switched on; no acknowledgement is necessary.) p 2080[7] = r 2139.7
      END_STRUCT;
      ActualSpeed : Int;   // Actual Speed 100%=4000 HEX = 16384 DEZ normalisation with p 2000 of the inverter
      ActualCurrent : Int;   // Actual Current 100%=4000 HEX = 16384 DEZ normalisation with p 2002 of the inverter
      ActualTorque : Int;   // Actual Torque 100%=4000 HEX = 16384 DEZ normalisation with p 2003 of the inverter
      AlarmCode : UInt;   // Actual alarm Code
      FaultCode : UInt;   // Actual fault Code
      XIST_A : DInt;   // Actual position value [LU]
      SpareWord9 : Int;   // Spare Word 9
      SpareWord10 : Int;   // Spare Word 10
      SpareWord11 : Int;   // Spare Word 11
   END_STRUCT;

END_TYPE

FUNCTION_BLOCK "FB_VfdSiemensCommissioning"
TITLE = FB_VFD_Siemens_Commissioning
{ S7_Optimized_Access := 'TRUE' }
AUTHOR : MHSE
VERSION : 3.2
// ATTRIBUTES
// AUTO_NUMBER = True
// BLOCK_NUMBER = 38
// END_ATTRIBUTES
   VAR_INPUT
      ihw_SinaParamHardwareId { ExternalAccessible := 'False'; ExternalVisible := 'False'; ExternalWritable := 'False'} : HW_IO := 0;   // Device hardware ID
      iUDT_MotorConfig { ExternalAccessible := 'False'; ExternalVisible := 'False'; ExternalWritable := 'False'} : "UDT_MotorData";   // Motor nad VFD parameters
      ix_Enable { ExternalAccessible := 'False'; ExternalVisible := 'False'; ExternalWritable := 'False'} : Bool;   // Input enable signal
   END_VAR

   VAR_OUTPUT
      qx_Busy { ExternalAccessible := 'False'; ExternalVisible := 'False'; ExternalWritable := 'False'} : Bool;   // Parametrization in progress
      qx_Done { ExternalAccessible := 'False'; ExternalVisible := 'False'; ExternalWritable := 'False'} : Bool;   // Parametrization done
      qx_Error { ExternalAccessible := 'False'; ExternalVisible := 'False'; ExternalWritable := 'False'} : Bool;   // Parametrization error
      qx_StartMeasuring { ExternalAccessible := 'False'; ExternalVisible := 'False'; ExternalWritable := 'False'} : Bool;   // Start measuring
   END_VAR

   VAR_IN_OUT
      iqx_GoToNextStep { ExternalAccessible := 'False'; ExternalVisible := 'False'; ExternalWritable := 'False'} : Bool;   // Go to next step
   END_VAR

